LIN {X 0,Y 519.821,Z 406.729,A -85,B 0,C 180,E1 -4932.29,E2 -4932.29} C_VEL
LIN {X 0,Y 519.302,Z 420.302,A -85,B 0,C 180,E1 -4933.084,E2 -4933.084} C_VEL
LIN {X 0,Y 518.746,Z 433.349,A -85,B 0,C 180,E1 -4934.021,E2 -4934.021} C_VEL
LIN {X 0,Y 518.217,Z 445.385,A -85,B 0,C 180,E1 -4935.067,E2 -4935.067} C_VEL
LIN {X 0,Y 517.729,Z 456.81,A -85,B 0,C 180,E1 -4936.257,E2 -4936.257} C_VEL
LIN {X 0,Y 517.347,Z 466.418,A -85,B 0,C 180,E1 -4937.446,E2 -4937.446} C_VEL
LIN {X 0,Y 517.02,Z 475.827,A -85,B 0,C 180,E1 -4938.831,E2 -4938.831} C_VEL
LIN {X 0,Y 516.707,Z 483.661,A -85,B 0,C 180,E1 -4940.211,E2 -4940.211} C_VEL
LIN {X 0,Y 516.511,Z 490.966,A -85,B 0,C 180,E1 -4941.786,E2 -4941.786} C_VEL
LIN {X 0,Y 516.372,Z 497.212,A -85,B 0,C 180,E1 -4943.493,E2 -4943.493} C_VEL
LIN {X 0,Y 516.373,Z 500.263,A -85,B 0,C 180,E1 -4944.533,E2 -4944.533} C_VEL
LIN {X 0,Y 516.308,Z 503.797,A -85,B 0,C 180,E1 -4946.097,E2 -4946.097} C_VEL
LIN {X 0,Y 516.259,Z 506.138,A -85,B 0,C 180,E1 -4947.659,E2 -4947.659} C_VEL
LIN {X 0,Y 516.156,Z 507.337,A -85,B 0,C 180,E1 -4949.22,E2 -4949.22} C_VEL
LIN {X 0,Y 516.157,Z 507.356,A -85,B 0,C 180,E1 -4950.78,E2 -4950.78} C_VEL
LIN {X 0,Y 516.259,Z 506.235,A -85,B 0,C 180,E1 -4952.34,E2 -4952.34} C_VEL
LIN {X 0,Y 516.308,Z 503.97,A -85,B 0,C 180,E1 -4953.902,E2 -4953.902} C_VEL
LIN {X 0,Y 516.369,Z 500.509,A -85,B 0,C 180,E1 -4955.467,E2 -4955.467} C_VEL
LIN {X 0,Y 516.392,Z 495.769,A -85,B 0,C 180,E1 -4957.035,E2 -4957.035} C_VEL
LIN {X 0,Y 516.541,Z 489.713,A -85,B 0,C 180,E1 -4958.607,E2 -4958.607} C_VEL
LIN {X 0,Y 516.758,Z 482.087,A -85,B 0,C 180,E1 -4960.183,E2 -4960.183} C_VEL
LIN {X 0,Y 517.014,Z 473.951,A -85,B 0,C 180,E1 -4961.566,E2 -4961.566} C_VEL
LIN {X 0,Y 517.423,Z 464.143,A -85,B 0,C 180,E1 -4962.95,E2 -4962.95} C_VEL
LIN {X 0,Y 517.829,Z 454.081,A -85,B 0,C 180,E1 -4964.14,E2 -4964.14} C_VEL
LIN {X 0,Y 518.306,Z 442.542,A -85,B 0,C 180,E1 -4965.289,E2 -4965.289} C_VEL
LIN {X 0,Y 518.904,Z 430.325,A -85,B 0,C 180,E1 -4966.301,E2 -4966.301} C_VEL
LIN {X 0,Y 519.365,Z 418.57,A -85,B 0,C 180,E1 -4967.116,E2 -4967.116} C_VEL
LIN {X 0,Y 519.835,Z 404.548,A -85,B 0,C 180,E1 -4967.913,E2 -4967.913} C_VEL
LIN {X 0,Y 520.354,Z 389.292,A -85,B 0,C 180,E1 -4968.583,E2 -4968.583} C_VEL
LIN {X 0,Y 520.704,Z 373.976,A -85,B 0,C 180,E1 -4969.078,E2 -4969.078} C_VEL
LIN {X 0,Y 520.233,Z 370.683,A -85,B 0,C 180,E1 -4969.188,E2 -4969.188} C_VEL
LIN {X 0,Y 516.92,Z 358.729,A -85,B 0,C 180,E1 -4969.566,E2 -4969.566} C_VEL
LIN {X 0,Y 516.34,Z 356.363,A -85,B 0,C 180,E1 -4969.649,E2 -4969.649} C_VEL
LIN {X 0,Y 516.364,Z 353.469,A -85,B 0,C 180,E1 -4972.401,E2 -4972.401} C_VEL
LIN {X 0,Y 516.389,Z 350.798,A -85,B 0,C 180,E1 -4974.955,E2 -4974.955} C_VEL
LIN {X 0,Y 516.469,Z 348.145,A -85,B 0,C 180,E1 -4977.559,E2 -4977.559} C_VEL
LIN {X 0,Y 516.495,Z 345.564,A -85,B 0,C 180,E1 -4980.229,E2 -4980.229} C_VEL
LIN {X 0,Y 516.579,Z 342.965,A -85,B 0,C 180,E1 -4982.969,E2 -4982.969} C_VEL
LIN {X 0,Y 516.601,Z 340.308,A -85,B 0,C 180,E1 -4985.801,E2 -4985.801} C_VEL
LIN {X 0,Y 516.629,Z 337.612,A -85,B 0,C 180,E1 -4988.738,E2 -4988.738} C_VEL
LIN {X 0,Y 516.66,Z 336.757,A -85,B 0,C 180,E1 -4989.741,E2 -4989.741} C_VEL
LIN {X 0,Y 516.848,Z 336.729,A -85,B 0,C 180,E1 -4991.781,E2 -4991.781} C_VEL
LIN {X 0,Y 516.922,Z 336.72,A -85,B 0,C 180,E1 -4995.01,E2 -4995.01} C_VEL
LIN {X 0,Y 516.916,Z 336.72,A -85,B 0,C 180,E1 -4998.398,E2 -4998.398} C_VEL
LIN {X 0,Y 516.882,Z 336.724,A -85,B 0,C 180,E1 -5001.284,E2 -5001.284} C_VEL
LIN {X 0,Y 516.891,Z 336.723,A -85,B 0,C 180,E1 -5004.221,E2 -5004.221} C_VEL
LIN {X 0,Y 516.895,Z 336.72,A -85,B 0,C 180,E1 -5007.053,E2 -5007.053} C_VEL
LIN {X 0,Y 516.901,Z 336.727,A -85,B 0,C 180,E1 -5009.797,E2 -5009.797} C_VEL
LIN {X 0,Y 516.929,Z 336.716,A -85,B 0,C 180,E1 -5012.467,E2 -5012.467} C_VEL
LIN {X 0,Y 516.911,Z 336.719,A -85,B 0,C 180,E1 -5015.072,E2 -5015.072} C_VEL
LIN {X 0,Y 516.885,Z 336.721,A -85,B 0,C 180,E1 -5018.462,E2 -5018.462} C_VEL
LIN {X 0,Y 516.904,Z 336.719,A -85,B 0,C 180,E1 -5020.955,E2 -5020.955} C_VEL
LIN {X 0,Y 516.916,Z 336.724,A -85,B 0,C 180,E1 -5023.41,E2 -5023.41} C_VEL
LIN {X 0,Y 516.894,Z 336.718,A -85,B 0,C 180,E1 -5025.834,E2 -5025.834} C_VEL
LIN {X 0,Y 517.003,Z 336.71,A -85,B 0,C 180,E1 -5028.234,E2 -5028.234} C_VEL
LIN {X 0,Y 516.969,Z 336.714,A -85,B 0,C 180,E1 -5031.4,E2 -5031.4} C_VEL
LIN {X 0,Y 517.011,Z 336.709,A -85,B 0,C 180,E1 -5033.757,E2 -5033.757} C_VEL
LIN {X 0,Y 517.082,Z 336.7,A -85,B 0,C 180,E1 -5037.663,E2 -5037.663} C_VEL
LIN {X 0,Y 517.093,Z 336.698,A -85,B 0,C 180,E1 -5040.779,E2 -5040.779} C_VEL
LIN {X 0,Y 517.014,Z 336.711,A -85,B 0,C 180,E1 -5043.117,E2 -5043.117} C_VEL
LIN {X 0,Y 517.009,Z 336.713,A -85,B 0,C 180,E1 -5046.243,E2 -5046.243} C_VEL
LIN {X 0,Y 516.952,Z 336.72,A -85,B 0,C 180,E1 -5049.389,E2 -5049.389} C_VEL
LIN {X 0,Y 516.955,Z 336.715,A -85,B 0,C 180,E1 -5051.81,E2 -5051.81} C_VEL
LIN {X 0,Y 516.942,Z 336.718,A -85,B 0,C 180,E1 -5055.147,E2 -5055.147} C_VEL
LIN {X 0,Y 516.923,Z 336.72,A -85,B 0,C 180,E1 -5058.222,E2 -5058.222} C_VEL
LIN {X 0,Y 516.91,Z 336.72,A -85,B 0,C 180,E1 -5060.701,E2 -5060.701} C_VEL
LIN {X 0,Y 516.909,Z 336.722,A -85,B 0,C 180,E1 -5064.072,E2 -5064.072} C_VEL
LIN {X 0,Y 516.924,Z 336.72,A -85,B 0,C 180,E1 -5066.658,E2 -5066.658} C_VEL
LIN {X 0,Y 516.918,Z 336.722,A -85,B 0,C 180,E1 -5069.526,E2 -5069.526} C_VEL
LIN {X 0,Y 516.899,Z 336.724,A -85,B 0,C 180,E1 -5072.544,E2 -5072.544} C_VEL
LIN {X 0,Y 516.881,Z 336.728,A -85,B 0,C 180,E1 -5075.333,E2 -5075.333} C_VEL
LIN {X 0,Y 516.88,Z 336.727,A -85,B 0,C 180,E1 -5077.944,E2 -5077.944} C_VEL
LIN {X 0,Y 516.884,Z 336.726,A -85,B 0,C 180,E1 -5080.742,E2 -5080.742} C_VEL
LIN {X 0,Y 516.882,Z 336.724,A -85,B 0,C 180,E1 -5082.831,E2 -5082.831} C_VEL
LIN {X 0,Y 516.924,Z 336.727,A -85,B 0,C 180,E1 -5085.011,E2 -5085.011} C_VEL
LIN {X 0,Y 517.783,Z 342.257,A -85,B 0,C 180,E1 -5087.789,E2 -5087.789} C_VEL
LIN {X 0,Y 517.985,Z 345.864,A -85,B 0,C 180,E1 -5089.447,E2 -5089.447} C_VEL
LIN {X 0,Y 517.741,Z 352.598,A -85,B 0,C 180,E1 -5092.35,E2 -5092.35} C_VEL
LIN {X 0,Y 517.609,Z 357.962,A -85,B 0,C 180,E1 -5094.554,E2 -5094.554} C_VEL
LIN {X 0,Y 517.413,Z 365.096,A -85,B 0,C 180,E1 -5097.367,E2 -5097.367} C_VEL
LIN {X 0,Y 517.242,Z 373.131,A -85,B 0,C 180,E1 -5100.412,E2 -5100.412} C_VEL
LIN {X 0,Y 517.066,Z 381.047,A -85,B 0,C 180,E1 -5103.35,E2 -5103.35} C_VEL
LIN {X 0,Y 516.871,Z 389.351,A -85,B 0,C 180,E1 -5106.352,E2 -5106.352} C_VEL
LIN {X 0,Y 516.77,Z 397.674,A -85,B 0,C 180,E1 -5109.293,E2 -5109.293} C_VEL
LIN {X 0,Y 516.703,Z 400.834,A -85,B 0,C 180,E1 -5110.381,E2 -5110.381} C_VEL
LIN {X 0,Y 520.44,Z 417.085,A -85,B 0,C 180,E1 -5110.825,E2 -5110.825} C_VEL
LIN {X 0,Y 520.664,Z 420.573,A -85,B 0,C 180,E1 -5110.919,E2 -5110.919} C_VEL
LIN {X 0,Y 520.288,Z 434.02,A -85,B 0,C 180,E1 -5111.32,E2 -5111.32} C_VEL
LIN {X 0,Y 519.885,Z 449.136,A -85,B 0,C 180,E1 -5111.936,E2 -5111.936} C_VEL
LIN {X 0,Y 519.372,Z 463.303,A -85,B 0,C 180,E1 -5112.681,E2 -5112.681} C_VEL
LIN {X 0,Y 518.84,Z 477.112,A -85,B 0,C 180,E1 -5113.585,E2 -5113.585} C_VEL
LIN {X 0,Y 518.397,Z 489.137,A -85,B 0,C 180,E1 -5114.542,E2 -5114.542} C_VEL
LIN {X 0,Y 517.857,Z 500.982,A -85,B 0,C 180,E1 -5115.66,E2 -5115.66} C_VEL
LIN {X 0,Y 517.47,Z 511.579,A -85,B 0,C 180,E1 -5116.851,E2 -5116.851} C_VEL
LIN {X 0,Y 517.012,Z 521.94,A -85,B 0,C 180,E1 -5118.235,E2 -5118.235} C_VEL
LIN {X 0,Y 516.89,Z 529.417,A -85,B 0,C 180,E1 -5119.423,E2 -5119.423} C_VEL
LIN {X 0,Y 516.637,Z 535.751,A -85,B 0,C 180,E1 -5120.605,E2 -5120.605} C_VEL
LIN {X 0,Y 516.462,Z 542.701,A -85,B 0,C 180,E1 -5122.179,E2 -5122.179} C_VEL
LIN {X 0,Y 516.36,Z 548.163,A -85,B 0,C 180,E1 -5123.749,E2 -5123.749} C_VEL
LIN {X 0,Y 516.238,Z 552.291,A -85,B 0,C 180,E1 -5125.315,E2 -5125.315} C_VEL
LIN {X 0,Y 516.272,Z 555.184,A -85,B 0,C 180,E1 -5126.879,E2 -5126.879} C_VEL
LIN {X 0,Y 516.189,Z 556.909,A -85,B 0,C 180,E1 -5128.44,E2 -5128.44} C_VEL
LIN {X 0,Y 516.151,Z 557.5,A -85,B 0,C 180,E1 -5130,E2 -5130} C_VEL
LIN {X 0,Y 516.189,Z 556.906,A -85,B 0,C 180,E1 -5131.561,E2 -5131.561} C_VEL
LIN {X 0,Y 516.272,Z 555.178,A -85,B 0,C 180,E1 -5133.122,E2 -5133.122} C_VEL
LIN {X 0,Y 516.238,Z 552.287,A -85,B 0,C 180,E1 -5134.686,E2 -5134.686} C_VEL
LIN {X 0,Y 516.376,Z 548.164,A -85,B 0,C 180,E1 -5136.251,E2 -5136.251} C_VEL
LIN {X 0,Y 516.463,Z 542.699,A -85,B 0,C 180,E1 -5137.821,E2 -5137.821} C_VEL
LIN {X 0,Y 516.638,Z 535.741,A -85,B 0,C 180,E1 -5139.395,E2 -5139.395} C_VEL
LIN {X 0,Y 516.911,Z 528.287,A -85,B 0,C 180,E1 -5140.775,E2 -5140.775} C_VEL
LIN {X 0,Y 517.138,Z 519.473,A -85,B 0,C 180,E1 -5142.121,E2 -5142.121} C_VEL
LIN {X 0,Y 517.536,Z 509.929,A -85,B 0,C 180,E1 -5143.348,E2 -5143.348} C_VEL
LIN {X 0,Y 517.917,Z 499.008,A -85,B 0,C 180,E1 -5144.539,E2 -5144.539} C_VEL
LIN {X 0,Y 518.445,Z 487.256,A -85,B 0,C 180,E1 -5145.617,E2 -5145.617} C_VEL
LIN {X 0,Y 518.952,Z 474.093,A -85,B 0,C 180,E1 -5146.624,E2 -5146.624} C_VEL
LIN {X 0,Y 519.491,Z 459.731,A -85,B 0,C 180,E1 -5147.519,E2 -5147.519} C_VEL
LIN {X 0,Y 520.048,Z 444.783,A -85,B 0,C 180,E1 -5148.254,E2 -5148.254} C_VEL
LIN {X 0,Y 520.425,Z 429.866,A -85,B 0,C 180,E1 -5148.814,E2 -5148.814} C_VEL
LIN {X 0,Y 520.592,Z 417.655,A -85,B 0,C 180,E1 -5149.157,E2 -5149.157} C_VEL
LIN {X 0,Y 516.706,Z 400.814,A -85,B 0,C 180,E1 -5149.626,E2 -5149.626} C_VEL
LIN {X 0,Y 516.833,Z 392.896,A -85,B 0,C 180,E1 -5152.38,E2 -5152.38} C_VEL
LIN {X 0,Y 517.025,Z 383.43,A -85,B 0,C 180,E1 -5155.784,E2 -5155.784} C_VEL
LIN {X 0,Y 517.201,Z 375.092,A -85,B 0,C 180,E1 -5158.842,E2 -5158.842} C_VEL
LIN {X 0,Y 517.373,Z 366.731,A -85,B 0,C 180,E1 -5161.991,E2 -5161.991} C_VEL
LIN {X 0,Y 517.517,Z 359.618,A -85,B 0,C 180,E1 -5164.776,E2 -5164.776} C_VEL
LIN {X 0,Y 517.741,Z 352.555,A -85,B 0,C 180,E1 -5167.651,E2 -5167.651} C_VEL
LIN {X 0,Y 517.907,Z 346.893,A -85,B 0,C 180,E1 -5170.085,E2 -5170.085} C_VEL
LIN {X 0,Y 517.896,Z 343.265,A -85,B 0,C 180,E1 -5171.724,E2 -5171.724} C_VEL
LIN {X 0,Y 517.082,Z 337.701,A -85,B 0,C 180,E1 -5174.475,E2 -5174.475} C_VEL
LIN {X 0,Y 516.916,Z 336.724,A -85,B 0,C 180,E1 -5175.009,E2 -5175.009} C_VEL
LIN {X 0,Y 516.915,Z 336.723,A -85,B 0,C 180,E1 -5178.399,E2 -5178.399} C_VEL
LIN {X 0,Y 516.884,Z 336.727,A -85,B 0,C 180,E1 -5181.284,E2 -5181.284} C_VEL
LIN {X 0,Y 516.894,Z 336.725,A -85,B 0,C 180,E1 -5184.222,E2 -5184.222} C_VEL
LIN {X 0,Y 516.897,Z 336.723,A -85,B 0,C 180,E1 -5187.053,E2 -5187.053} C_VEL
LIN {X 0,Y 516.895,Z 336.724,A -85,B 0,C 180,E1 -5189.797,E2 -5189.797} C_VEL
LIN {X 0,Y 516.931,Z 336.723,A -85,B 0,C 180,E1 -5192.468,E2 -5192.468} C_VEL
LIN {X 0,Y 516.911,Z 336.722,A -85,B 0,C 180,E1 -5195.072,E2 -5195.072} C_VEL
LIN {X 0,Y 516.889,Z 336.728,A -85,B 0,C 180,E1 -5198.463,E2 -5198.463} C_VEL
LIN {X 0,Y 516.906,Z 336.721,A -85,B 0,C 180,E1 -5200.955,E2 -5200.955} C_VEL
LIN {X 0,Y 516.917,Z 336.722,A -85,B 0,C 180,E1 -5203.41,E2 -5203.41} C_VEL
LIN {X 0,Y 516.899,Z 336.725,A -85,B 0,C 180,E1 -5205.834,E2 -5205.834} C_VEL
LIN {X 0,Y 516.969,Z 336.714,A -85,B 0,C 180,E1 -5208.234,E2 -5208.234} C_VEL
LIN {X 0,Y 516.972,Z 336.713,A -85,B 0,C 180,E1 -5211.4,E2 -5211.4} C_VEL
LIN {X 0,Y 517.013,Z 336.712,A -85,B 0,C 180,E1 -5213.757,E2 -5213.757} C_VEL
LIN {X 0,Y 517.087,Z 336.698,A -85,B 0,C 180,E1 -5217.663,E2 -5217.663} C_VEL
LIN {X 0,Y 517.098,Z 336.697,A -85,B 0,C 180,E1 -5220.779,E2 -5220.779} C_VEL
LIN {X 0,Y 517.017,Z 336.708,A -85,B 0,C 180,E1 -5223.117,E2 -5223.117} C_VEL
LIN {X 0,Y 517.015,Z 336.707,A -85,B 0,C 180,E1 -5226.243,E2 -5226.243} C_VEL
LIN {X 0,Y 516.957,Z 336.715,A -85,B 0,C 180,E1 -5229.389,E2 -5229.389} C_VEL
LIN {X 0,Y 516.956,Z 336.714,A -85,B 0,C 180,E1 -5231.807,E2 -5231.807} C_VEL
LIN {X 0,Y 516.948,Z 336.719,A -85,B 0,C 180,E1 -5235.146,E2 -5235.146} C_VEL
LIN {X 0,Y 516.929,Z 336.719,A -85,B 0,C 180,E1 -5238.222,E2 -5238.222} C_VEL
LIN {X 0,Y 516.916,Z 336.711,A -85,B 0,C 180,E1 -5240.701,E2 -5240.701} C_VEL
LIN {X 0,Y 516.894,Z 336.726,A -85,B 0,C 180,E1 -5244.073,E2 -5244.073} C_VEL
LIN {X 0,Y 516.928,Z 336.714,A -85,B 0,C 180,E1 -5246.658,E2 -5246.658} C_VEL
LIN {X 0,Y 516.915,Z 336.719,A -85,B 0,C 180,E1 -5249.524,E2 -5249.524} C_VEL
LIN {X 0,Y 516.899,Z 336.719,A -85,B 0,C 180,E1 -5252.543,E2 -5252.543} C_VEL
LIN {X 0,Y 516.883,Z 336.724,A -85,B 0,C 180,E1 -5255.332,E2 -5255.332} C_VEL
LIN {X 0,Y 516.885,Z 336.729,A -85,B 0,C 180,E1 -5257.943,E2 -5257.943} C_VEL
LIN {X 0,Y 516.888,Z 336.727,A -85,B 0,C 180,E1 -5260.741,E2 -5260.741} C_VEL
LIN {X 0,Y 516.887,Z 336.726,A -85,B 0,C 180,E1 -5262.831,E2 -5262.831} C_VEL
LIN {X 0,Y 516.926,Z 336.72,A -85,B 0,C 180,E1 -5265.01,E2 -5265.01} C_VEL
LIN {X 0,Y 516.851,Z 336.731,A -85,B 0,C 180,E1 -5268.218,E2 -5268.218} C_VEL
LIN {X 0,Y 516.672,Z 336.776,A -85,B 0,C 180,E1 -5270.292,E2 -5270.292} C_VEL
LIN {X 0,Y 515.975,Z 337.328,A -85,B 0,C 180,E1 -5270.939,E2 -5270.939} C_VEL
LIN {X 0,Y 513.098,Z 338.557,A -85,B 0,C 180,E1 -5271.987,E2 -5271.987} C_VEL
LIN {X 0,Y 510.678,Z 339.577,A -85,B 0,C 180,E1 -5272.83,E2 -5272.83} C_VEL
LIN {X 0,Y 509.635,Z 340.277,A -85,B 0,C 180,E1 -5273.482,E2 -5273.482} C_VEL
LIN {X 0,Y 509.547,Z 340.487,A -85,B 0,C 180,E1 -5273.703,E2 -5273.703} C_VEL
LIN {X 0,Y 509.517,Z 343.074,A -85,B 0,C 180,E1 -5276.513,E2 -5276.513} C_VEL
LIN {X 0,Y 509.437,Z 345.693,A -85,B 0,C 180,E1 -5279.307,E2 -5279.307} C_VEL
LIN {X 0,Y 509.404,Z 348.283,A -85,B 0,C 180,E1 -5282.025,E2 -5282.025} C_VEL
LIN {X 0,Y 509.356,Z 350.915,A -85,B 0,C 180,E1 -5284.676,E2 -5284.676} C_VEL
LIN {X 0,Y 509.299,Z 353.973,A -85,B 0,C 180,E1 -5287.602,E2 -5287.602} C_VEL
LIN {X 0,Y 509.284,Z 356.802,A -85,B 0,C 180,E1 -5290.177,E2 -5290.177} C_VEL
LIN {X 0,Y 513.395,Z 371.414,A -85,B 0,C 180,E1 -5290.646,E2 -5290.646} C_VEL
LIN {X 0,Y 513.96,Z 374.193,A -85,B 0,C 180,E1 -5290.748,E2 -5290.748} C_VEL
LIN {X 0,Y 513.663,Z 388.561,A -85,B 0,C 180,E1 -5291.213,E2 -5291.213} C_VEL
LIN {X 0,Y 513.16,Z 403.143,A -85,B 0,C 180,E1 -5291.846,E2 -5291.846} C_VEL
LIN {X 0,Y 512.634,Z 417.516,A -85,B 0,C 180,E1 -5292.651,E2 -5292.651} C_VEL
LIN {X 0,Y 512.067,Z 430.567,A -85,B 0,C 180,E1 -5293.556,E2 -5293.556} C_VEL
LIN {X 0,Y 511.549,Z 441.99,A -85,B 0,C 180,E1 -5294.507,E2 -5294.507} C_VEL
LIN {X 0,Y 510.97,Z 453.632,A -85,B 0,C 180,E1 -5295.666,E2 -5295.666} C_VEL
LIN {X 0,Y 510.518,Z 463.777,A -85,B 0,C 180,E1 -5296.871,E2 -5296.871} C_VEL
LIN {X 0,Y 510.087,Z 473.286,A -85,B 0,C 180,E1 -5298.211,E2 -5298.211} C_VEL
LIN {X 0,Y 509.828,Z 480.826,A -85,B 0,C 180,E1 -5299.475,E2 -5299.475} C_VEL
LIN {X 0,Y 509.584,Z 487.865,A -85,B 0,C 180,E1 -5300.874,E2 -5300.874} C_VEL
LIN {X 0,Y 509.39,Z 494.393,A -85,B 0,C 180,E1 -5302.468,E2 -5302.468} C_VEL
LIN {X 0,Y 509.313,Z 499.494,A -85,B 0,C 180,E1 -5304.059,E2 -5304.059} C_VEL
LIN {X 0,Y 509.159,Z 502.438,A -85,B 0,C 180,E1 -5305.249,E2 -5305.249} C_VEL
LIN {X 0,Y 509.188,Z 505.316,A -85,B 0,C 180,E1 -5306.835,E2 -5306.835} C_VEL
LIN {X 0,Y 509.11,Z 507.057,A -85,B 0,C 180,E1 -5308.418,E2 -5308.418} C_VEL
LIN {X 0,Y 509.063,Z 507.667,A -85,B 0,C 180,E1 -5310,E2 -5310} C_VEL
LIN {X 0,Y 509.111,Z 507.113,A -85,B 0,C 180,E1 -5311.582,E2 -5311.582} C_VEL
LIN {X 0,Y 509.189,Z 505.448,A -85,B 0,C 180,E1 -5313.165,E2 -5313.165} C_VEL
LIN {X 0,Y 509.158,Z 502.641,A -85,B 0,C 180,E1 -5314.75,E2 -5314.75} C_VEL
LIN {X 0,Y 509.26,Z 498.613,A -85,B 0,C 180,E1 -5316.338,E2 -5316.338} C_VEL
LIN {X 0,Y 509.412,Z 493.269,A -85,B 0,C 180,E1 -5317.93,E2 -5317.93} C_VEL
LIN {X 0,Y 509.614,Z 486.458,A -85,B 0,C 180,E1 -5319.525,E2 -5319.525} C_VEL
LIN {X 0,Y 509.96,Z 477.948,A -85,B 0,C 180,E1 -5321.124,E2 -5321.124} C_VEL
LIN {X 0,Y 510.285,Z 468.902,A -85,B 0,C 180,E1 -5322.528,E2 -5322.528} C_VEL
LIN {X 0,Y 510.698,Z 459.668,A -85,B 0,C 180,E1 -5323.732,E2 -5323.732} C_VEL
LIN {X 0,Y 511.237,Z 447.728,A -85,B 0,C 180,E1 -5325.039,E2 -5325.039} C_VEL
LIN {X 0,Y 511.86,Z 435.522,A -85,B 0,C 180,E1 -5326.142,E2 -5326.142} C_VEL
LIN {X 0,Y 512.447,Z 422.046,A -85,B 0,C 180,E1 -5327.149,E2 -5327.149} C_VEL
LIN {X 0,Y 512.959,Z 408.785,A -85,B 0,C 180,E1 -5327.955,E2 -5327.955} C_VEL
LIN {X 0,Y 513.493,Z 394.989,A -85,B 0,C 180,E1 -5328.619,E2 -5328.619} C_VEL
LIN {X 0,Y 513.869,Z 380.906,A -85,B 0,C 180,E1 -5329.142,E2 -5329.142} C_VEL
LIN {X 0,Y 513.814,Z 373.203,A -85,B 0,C 180,E1 -5329.376,E2 -5329.376} C_VEL
LIN {X 0,Y 510.626,Z 361.408,A -85,B 0,C 180,E1 -5329.776,E2 -5329.776} C_VEL
LIN {X 0,Y 509.297,Z 356.686,A -85,B 0,C 180,E1 -5329.92,E2 -5329.92} C_VEL
LIN {X 0,Y 509.289,Z 353.731,A -85,B 0,C 180,E1 -5332.73,E2 -5332.73} C_VEL
LIN {X 0,Y 509.353,Z 351.009,A -85,B 0,C 180,E1 -5335.323,E2 -5335.323} C_VEL
LIN {X 0,Y 509.388,Z 348.368,A -85,B 0,C 180,E1 -5337.993,E2 -5337.993} C_VEL
LIN {X 0,Y 509.476,Z 345.302,A -85,B 0,C 180,E1 -5341.211,E2 -5341.211} C_VEL
LIN {X 0,Y 509.541,Z 342.55,A -85,B 0,C 180,E1 -5344.15,E2 -5344.15} C_VEL
LIN {X 0,Y 509.562,Z 340.045,A -85,B 0,C 180,E1 -5346.875,E2 -5346.875} C_VEL
LIN {X 0,Y 509.589,Z 337.733,A -85,B 0,C 180,E1 -5349.437,E2 -5349.437} C_VEL
LIN {X 0,Y 509.803,Z 337.605,A -85,B 0,C 180,E1 -5351.89,E2 -5351.89} C_VEL
LIN {X 0,Y 509.856,Z 337.603,A -85,B 0,C 180,E1 -5354.668,E2 -5354.668} C_VEL
LIN {X 0,Y 509.857,Z 337.6,A -85,B 0,C 180,E1 -5358.103,E2 -5358.103} C_VEL
LIN {X 0,Y 509.847,Z 337.605,A -85,B 0,C 180,E1 -5360.647,E2 -5360.647} C_VEL
LIN {X 0,Y 509.836,Z 337.606,A -85,B 0,C 180,E1 -5363.648,E2 -5363.648} C_VEL
LIN {X 0,Y 509.861,Z 337.599,A -85,B 0,C 180,E1 -5366.539,E2 -5366.539} C_VEL
LIN {X 0,Y 509.85,Z 337.6,A -85,B 0,C 180,E1 -5369.334,E2 -5369.334} C_VEL
LIN {X 0,Y 509.894,Z 337.59,A -85,B 0,C 180,E1 -5372.054,E2 -5372.054} C_VEL
LIN {X 0,Y 509.877,Z 337.597,A -85,B 0,C 180,E1 -5374.704,E2 -5374.704} C_VEL
LIN {X 0,Y 509.855,Z 337.601,A -85,B 0,C 180,E1 -5377.449,E2 -5377.449} C_VEL
LIN {X 0,Y 509.915,Z 337.583,A -85,B 0,C 180,E1 -5379.845,E2 -5379.845} C_VEL
LIN {X 0,Y 509.886,Z 337.597,A -85,B 0,C 180,E1 -5383.175,E2 -5383.175} C_VEL
LIN {X 0,Y 509.863,Z 337.593,A -85,B 0,C 180,E1 -5385.634,E2 -5385.634} C_VEL
LIN {X 0,Y 509.921,Z 337.589,A -85,B 0,C 180,E1 -5388.875,E2 -5388.875} C_VEL
LIN {X 0,Y 509.95,Z 337.587,A -85,B 0,C 180,E1 -5392.078,E2 -5392.078} C_VEL
LIN {X 0,Y 509.982,Z 337.585,A -85,B 0,C 180,E1 -5394.464,E2 -5394.464} C_VEL
LIN {X 0,Y 510.053,Z 337.576,A -85,B 0,C 180,E1 -5397.631,E2 -5397.631} C_VEL
LIN {X 0,Y 510.063,Z 337.574,A -85,B 0,C 180,E1 -5400.789,E2 -5400.789} C_VEL
LIN {X 0,Y 509.956,Z 337.59,A -85,B 0,C 180,E1 -5403.16,E2 -5403.16} C_VEL
LIN {X 0,Y 509.977,Z 337.589,A -85,B 0,C 180,E1 -5406.33,E2 -5406.33} C_VEL
LIN {X 0,Y 509.914,Z 337.592,A -85,B 0,C 180,E1 -5408.72,E2 -5408.72} C_VEL
LIN {X 0,Y 509.903,Z 337.594,A -85,B 0,C 180,E1 -5411.932,E2 -5411.932} C_VEL
LIN {X 0,Y 509.891,Z 337.597,A -85,B 0,C 180,E1 -5415.242,E2 -5415.242} C_VEL
LIN {X 0,Y 509.886,Z 337.595,A -85,B 0,C 180,E1 -5418.001,E2 -5418.001} C_VEL
LIN {X 0,Y 509.848,Z 337.6,A -85,B 0,C 180,E1 -5421.002,E2 -5421.002} C_VEL
LIN {X 0,Y 509.835,Z 337.603,A -85,B 0,C 180,E1 -5423.563,E2 -5423.563} C_VEL
LIN {X 0,Y 509.91,Z 337.596,A -85,B 0,C 180,E1 -5426.379,E2 -5426.379} C_VEL
LIN {X 0,Y 509.879,Z 337.599,A -85,B 0,C 180,E1 -5428.844,E2 -5428.844} C_VEL
LIN {X 0,Y 509.824,Z 337.604,A -85,B 0,C 180,E1 -5431.59,E2 -5431.59} C_VEL
LIN {X 0,Y 509.852,Z 337.601,A -85,B 0,C 180,E1 -5434.413,E2 -5434.413} C_VEL
LIN {X 0,Y 509.818,Z 337.605,A -85,B 0,C 180,E1 -5437.341,E2 -5437.341} C_VEL
LIN {X 0,Y 509.837,Z 337.604,A -85,B 0,C 180,E1 -5440.382,E2 -5440.382} C_VEL
LIN {X 0,Y 509.822,Z 337.604,A -85,B 0,C 180,E1 -5443.063,E2 -5443.063} C_VEL
LIN {X 0,Y 509.873,Z 337.71,A -85,B 0,C 180,E1 -5444.756,E2 -5444.756} C_VEL
LIN {X 0,Y 510.778,Z 343.299,A -85,B 0,C 180,E1 -5447.608,E2 -5447.608} C_VEL
LIN {X 0,Y 511.015,Z 346.574,A -85,B 0,C 180,E1 -5449.149,E2 -5449.149} C_VEL
LIN {X 0,Y 510.812,Z 352.471,A -85,B 0,C 180,E1 -5451.748,E2 -5451.748} C_VEL
LIN {X 0,Y 510.597,Z 359.462,A -85,B 0,C 180,E1 -5454.683,E2 -5454.683} C_VEL
LIN {X 0,Y 510.364,Z 367.762,A -85,B 0,C 180,E1 -5457.984,E2 -5457.984} C_VEL
LIN {X 0,Y 510.181,Z 376.111,A -85,B 0,C 180,E1 -5461.175,E2 -5461.175} C_VEL
LIN {X 0,Y 509.947,Z 384.411,A -85,B 0,C 180,E1 -5464.271,E2 -5464.271} C_VEL
LIN {X 0,Y 509.772,Z 393.14,A -85,B 0,C 180,E1 -5467.473,E2 -5467.473} C_VEL
LIN {X 0,Y 509.643,Z 400.435,A -85,B 0,C 180,E1 -5470.087,E2 -5470.087} C_VEL
LIN {X 0,Y 513.688,Z 418.149,A -85,B 0,C 180,E1 -5470.595,E2 -5470.595} C_VEL
LIN {X 0,Y 513.921,Z 420.916,A -85,B 0,C 180,E1 -5470.679,E2 -5470.679} C_VEL
LIN {X 0,Y 513.527,Z 434.316,A -85,B 0,C 180,E1 -5471.088,E2 -5471.088} C_VEL
LIN {X 0,Y 513.108,Z 448.787,A -85,B 0,C 180,E1 -5471.689,E2 -5471.689} C_VEL
LIN {X 0,Y 512.558,Z 462.953,A -85,B 0,C 180,E1 -5472.443,E2 -5472.443} C_VEL
LIN {X 0,Y 511.967,Z 476.618,A -85,B 0,C 180,E1 -5473.348,E2 -5473.348} C_VEL
LIN {X 0,Y 511.437,Z 489.463,A -85,B 0,C 180,E1 -5474.385,E2 -5474.385} C_VEL
LIN {X 0,Y 510.905,Z 500.63,A -85,B 0,C 180,E1 -5475.461,E2 -5475.461} C_VEL
LIN {X 0,Y 510.476,Z 511.227,A -85,B 0,C 180,E1 -5476.668,E2 -5476.668} C_VEL
LIN {X 0,Y 510.001,Z 521.589,A -85,B 0,C 180,E1 -5478.071,E2 -5478.071} C_VEL
LIN {X 0,Y 509.786,Z 530.216,A -85,B 0,C 180,E1 -5479.475,E2 -5479.475} C_VEL
LIN {X 0,Y 509.516,Z 537.391,A -85,B 0,C 180,E1 -5480.873,E2 -5480.873} C_VEL
LIN {X 0,Y 509.351,Z 544.053,A -85,B 0,C 180,E1 -5482.468,E2 -5482.468} C_VEL
LIN {X 0,Y 509.275,Z 549.268,A -85,B 0,C 180,E1 -5484.06,E2 -5484.06} C_VEL
LIN {X 0,Y 509.158,Z 552.277,A -85,B 0,C 180,E1 -5485.25,E2 -5485.25} C_VEL
LIN {X 0,Y 509.188,Z 555.183,A -85,B 0,C 180,E1 -5486.835,E2 -5486.835} C_VEL
LIN {X 0,Y 509.11,Z 556.909,A -85,B 0,C 180,E1 -5488.418,E2 -5488.418} C_VEL
LIN {X 0,Y 509.062,Z 557.5,A -85,B 0,C 180,E1 -5490,E2 -5490} C_VEL
LIN {X 0,Y 509.11,Z 556.906,A -85,B 0,C 180,E1 -5491.582,E2 -5491.582} C_VEL
LIN {X 0,Y 509.188,Z 555.177,A -85,B 0,C 180,E1 -5493.165,E2 -5493.165} C_VEL
LIN {X 0,Y 509.159,Z 552.274,A -85,B 0,C 180,E1 -5494.751,E2 -5494.751} C_VEL
LIN {X 0,Y 509.306,Z 548.094,A -85,B 0,C 180,E1 -5496.338,E2 -5496.338} C_VEL
LIN {X 0,Y 509.385,Z 542.545,A -85,B 0,C 180,E1 -5497.931,E2 -5497.931} C_VEL
LIN {X 0,Y 509.546,Z 535.488,A -85,B 0,C 180,E1 -5499.527,E2 -5499.527} C_VEL
LIN {X 0,Y 509.905,Z 526.716,A -85,B 0,C 180,E1 -5501.126,E2 -5501.126} C_VEL
LIN {X 0,Y 510.201,Z 517.396,A -85,B 0,C 180,E1 -5502.531,E2 -5502.531} C_VEL
LIN {X 0,Y 510.607,Z 507.929,A -85,B 0,C 180,E1 -5503.735,E2 -5503.735} C_VEL
LIN {X 0,Y 511.103,Z 495.661,A -85,B 0,C 180,E1 -5505.043,E2 -5505.043} C_VEL
LIN {X 0,Y 511.718,Z 483.163,A -85,B 0,C 180,E1 -5506.148,E2 -5506.148} C_VEL
LIN {X 0,Y 512.212,Z 470.869,A -85,B 0,C 180,E1 -5507.055,E2 -5507.055} C_VEL
LIN {X 0,Y 512.749,Z 457.605,A -85,B 0,C 180,E1 -5507.86,E2 -5507.86} C_VEL
LIN {X 0,Y 513.305,Z 443.025,A -85,B 0,C 180,E1 -5508.566,E2 -5508.566} C_VEL
LIN {X 0,Y 513.713,Z 428.753,A -85,B 0,C 180,E1 -5509.095,E2 -5509.095} C_VEL
LIN {X 0,Y 513.847,Z 418.782,A -85,B 0,C 180,E1 -5509.384,E2 -5509.384} C_VEL
LIN {X 0,Y 509.995,Z 402.5,A -85,B 0,C 180,E1 -5509.859,E2 -5509.859} C_VEL
LIN {X 0,Y 509.622,Z 400.449,A -85,B 0,C 180,E1 -5509.909,E2 -5509.909} C_VEL
LIN {X 0,Y 509.749,Z 392.638,A -85,B 0,C 180,E1 -5512.709,E2 -5512.709} C_VEL
LIN {X 0,Y 509.96,Z 384.4,A -85,B 0,C 180,E1 -5515.729,E2 -5515.729} C_VEL
LIN {X 0,Y 510.179,Z 376.071,A -85,B 0,C 180,E1 -5518.826,E2 -5518.826} C_VEL
LIN {X 0,Y 510.365,Z 367.721,A -85,B 0,C 180,E1 -5522.017,E2 -5522.017} C_VEL
LIN {X 0,Y 510.591,Z 359.445,A -85,B 0,C 180,E1 -5525.318,E2 -5525.318} C_VEL
LIN {X 0,Y 510.811,Z 352.184,A -85,B 0,C 180,E1 -5528.35,E2 -5528.35} C_VEL
LIN {X 0,Y 510.968,Z 346.552,A -85,B 0,C 180,E1 -5530.845,E2 -5530.845} C_VEL
LIN {X 0,Y 510.777,Z 343.268,A -85,B 0,C 180,E1 -5532.393,E2 -5532.393} C_VEL
LIN {X 0,Y 509.853,Z 337.599,A -85,B 0,C 180,E1 -5535.332,E2 -5535.332} C_VEL
LIN {X 0,Y 509.857,Z 337.603,A -85,B 0,C 180,E1 -5538.575,E2 -5538.575} C_VEL
LIN {X 0,Y 509.854,Z 337.605,A -85,B 0,C 180,E1 -5541.787,E2 -5541.787} C_VEL
LIN {X 0,Y 509.849,Z 337.605,A -85,B 0,C 180,E1 -5544.624,E2 -5544.624} C_VEL
LIN {X 0,Y 509.863,Z 337.601,A -85,B 0,C 180,E1 -5547.481,E2 -5547.481} C_VEL
LIN {X 0,Y 509.861,Z 337.599,A -85,B 0,C 180,E1 -5550.274,E2 -5550.274} C_VEL
LIN {X 0,Y 509.888,Z 337.596,A -85,B 0,C 180,E1 -5552.945,E2 -5552.945} C_VEL
LIN {X 0,Y 509.867,Z 337.602,A -85,B 0,C 180,E1 -5555.574,E2 -5555.574} C_VEL
LIN {X 0,Y 509.854,Z 337.6,A -85,B 0,C 180,E1 -5558.999,E2 -5558.999} C_VEL
LIN {X 0,Y 509.892,Z 337.596,A -85,B 0,C 180,E1 -5561.999,E2 -5561.999} C_VEL
LIN {X 0,Y 509.914,Z 337.596,A -85,B 0,C 180,E1 -5564.819,E2 -5564.819} C_VEL
LIN {X 0,Y 509.905,Z 337.595,A -85,B 0,C 180,E1 -5568.124,E2 -5568.124} C_VEL
LIN {X 0,Y 509.918,Z 337.592,A -85,B 0,C 180,E1 -5571.28,E2 -5571.28} C_VEL
LIN {X 0,Y 509.981,Z 337.588,A -85,B 0,C 180,E1 -5573.671,E2 -5573.671} C_VEL
LIN {X 0,Y 510.058,Z 337.574,A -85,B 0,C 180,E1 -5577.631,E2 -5577.631} C_VEL
LIN {X 0,Y 510.068,Z 337.572,A -85,B 0,C 180,E1 -5580.79,E2 -5580.79} C_VEL
LIN {X 0,Y 509.959,Z 337.587,A -85,B 0,C 180,E1 -5583.16,E2 -5583.16} C_VEL
LIN {X 0,Y 509.984,Z 337.583,A -85,B 0,C 180,E1 -5586.33,E2 -5586.33} C_VEL
LIN {X 0,Y 509.92,Z 337.594,A -85,B 0,C 180,E1 -5588.72,E2 -5588.72} C_VEL
LIN {X 0,Y 509.908,Z 337.589,A -85,B 0,C 180,E1 -5591.932,E2 -5591.932} C_VEL
LIN {X 0,Y 509.898,Z 337.596,A -85,B 0,C 180,E1 -5595.242,E2 -5595.242} C_VEL
LIN {X 0,Y 509.892,Z 337.598,A -85,B 0,C 180,E1 -5598.001,E2 -5598.001} C_VEL
LIN {X 0,Y 509.854,Z 337.593,A -85,B 0,C 180,E1 -5601.002,E2 -5601.002} C_VEL
LIN {X 0,Y 509.826,Z 337.602,A -85,B 0,C 180,E1 -5603.564,E2 -5603.564} C_VEL
LIN {X 0,Y 509.915,Z 337.587,A -85,B 0,C 180,E1 -5606.378,E2 -5606.378} C_VEL
LIN {X 0,Y 509.88,Z 337.598,A -85,B 0,C 180,E1 -5608.844,E2 -5608.844} C_VEL
LIN {X 0,Y 509.824,Z 337.606,A -85,B 0,C 180,E1 -5611.59,E2 -5611.59} C_VEL
LIN {X 0,Y 509.855,Z 337.596,A -85,B 0,C 180,E1 -5614.413,E2 -5614.413} C_VEL
LIN {X 0,Y 509.823,Z 337.604,A -85,B 0,C 180,E1 -5617.34,E2 -5617.34} C_VEL
LIN {X 0,Y 509.841,Z 337.602,A -85,B 0,C 180,E1 -5620.382,E2 -5620.382} C_VEL
LIN {X 0,Y 509.827,Z 337.604,A -85,B 0,C 180,E1 -5623.062,E2 -5623.062} C_VEL
LIN {X 0,Y 509.834,Z 337.606,A -85,B 0,C 180,E1 -5625.792,E2 -5625.792} C_VEL
LIN {X 0,Y 509.777,Z 337.615,A -85,B 0,C 180,E1 -5628.566,E2 -5628.566} C_VEL
LIN {X 0,Y 509.601,Z 337.7,A -85,B 0,C 180,E1 -5630.625,E2 -5630.625} C_VEL
LIN {X 0,Y 509.547,Z 340.487,A -85,B 0,C 180,E1 -5633.703,E2 -5633.703} C_VEL
LIN {X 0,Y 508.875,Z 341.159,A -85,B 0,C 180,E1 -5634.359,E2 -5634.359} C_VEL
LIN {X 0,Y 506.024,Z 342.437,A -85,B 0,C 180,E1 -5635.422,E2 -5635.422} C_VEL
LIN {X 0,Y 503.602,Z 343.472,A -85,B 0,C 180,E1 -5636.277,E2 -5636.277} C_VEL
LIN {X 0,Y 502.542,Z 344.18,A -85,B 0,C 180,E1 -5636.939,E2 -5636.939} C_VEL
LIN {X 0,Y 502.444,Z 344.392,A -85,B 0,C 180,E1 -5637.164,E2 -5637.164} C_VEL
LIN {X 0,Y 502.36,Z 347.18,A -85,B 0,C 180,E1 -5640.156,E2 -5640.156} C_VEL
LIN {X 0,Y 502.3,Z 349.394,A -85,B 0,C 180,E1 -5642.501,E2 -5642.501} C_VEL
LIN {X 0,Y 502.245,Z 352.34,A -85,B 0,C 180,E1 -5645.444,E2 -5645.444} C_VEL
LIN {X 0,Y 502.187,Z 355.723,A -85,B 0,C 180,E1 -5648.662,E2 -5648.662} C_VEL
LIN {X 0,Y 502.251,Z 357.282,A -85,B 0,C 180,E1 -5649.89,E2 -5649.89} C_VEL
LIN {X 0,Y 506.55,Z 371.981,A -85,B 0,C 180,E1 -5650.379,E2 -5650.379} C_VEL
LIN {X 0,Y 507.256,Z 376.124,A -85,B 0,C 180,E1 -5650.528,E2 -5650.528} C_VEL
LIN {X 0,Y 506.924,Z 390.567,A -85,B 0,C 180,E1 -5651.02,E2 -5651.02} C_VEL
LIN {X 0,Y 506.363,Z 405.477,A -85,B 0,C 180,E1 -5651.698,E2 -5651.698} C_VEL
LIN {X 0,Y 505.781,Z 419.447,A -85,B 0,C 180,E1 -5652.513,E2 -5652.513} C_VEL
LIN {X 0,Y 505.199,Z 432.206,A -85,B 0,C 180,E1 -5653.43,E2 -5653.43} C_VEL
LIN {X 0,Y 504.547,Z 444.337,A -85,B 0,C 180,E1 -5654.481,E2 -5654.481} C_VEL
LIN {X 0,Y 503.99,Z 455.756,A -85,B 0,C 180,E1 -5655.669,E2 -5655.669} C_VEL
LIN {X 0,Y 503.505,Z 465.658,A -85,B 0,C 180,E1 -5656.89,E2 -5656.89} C_VEL
LIN {X 0,Y 503.067,Z 475.32,A -85,B 0,C 180,E1 -5658.312,E2 -5658.312} C_VEL
LIN {X 0,Y 502.696,Z 483.37,A -85,B 0,C 180,E1 -5659.732,E2 -5659.732} C_VEL
LIN {X 0,Y 502.497,Z 490.002,A -85,B 0,C 180,E1 -5661.15,E2 -5661.15} C_VEL
LIN {X 0,Y 502.294,Z 496.148,A -85,B 0,C 180,E1 -5662.765,E2 -5662.765} C_VEL
LIN {X 0,Y 502.241,Z 500.89,A -85,B 0,C 180,E1 -5664.378,E2 -5664.378} C_VEL
LIN {X 0,Y 502.166,Z 504.369,A -85,B 0,C 180,E1 -5665.987,E2 -5665.987} C_VEL
LIN {X 0,Y 502.118,Z 506.672,A -85,B 0,C 180,E1 -5667.593,E2 -5667.593} C_VEL
LIN {X 0,Y 501.987,Z 507.857,A -85,B 0,C 180,E1 -5669.197,E2 -5669.197} C_VEL
LIN {X 0,Y 501.988,Z 507.876,A -85,B 0,C 180,E1 -5670.802,E2 -5670.802} C_VEL
LIN {X 0,Y 502.118,Z 506.765,A -85,B 0,C 180,E1 -5672.406,E2 -5672.406} C_VEL
LIN {X 0,Y 502.166,Z 504.535,A -85,B 0,C 180,E1 -5674.012,E2 -5674.012} C_VEL
LIN {X 0,Y 502.233,Z 501.126,A -85,B 0,C 180,E1 -5675.621,E2 -5675.621} C_VEL
LIN {X 0,Y 502.293,Z 496.459,A -85,B 0,C 180,E1 -5677.234,E2 -5677.234} C_VEL
LIN {X 0,Y 502.493,Z 490.404,A -85,B 0,C 180,E1 -5678.85,E2 -5678.85} C_VEL
LIN {X 0,Y 502.746,Z 482.778,A -85,B 0,C 180,E1 -5680.47,E2 -5680.47} C_VEL
LIN {X 0,Y 503.057,Z 474.697,A -85,B 0,C 180,E1 -5681.883,E2 -5681.883} C_VEL
LIN {X 0,Y 503.574,Z 464.831,A -85,B 0,C 180,E1 -5683.313,E2 -5683.313} C_VEL
LIN {X 0,Y 504.049,Z 454.767,A -85,B 0,C 180,E1 -5684.535,E2 -5684.535} C_VEL
LIN {X 0,Y 504.576,Z 443.722,A -85,B 0,C 180,E1 -5685.667,E2 -5685.667} C_VEL
LIN {X 0,Y 505.22,Z 432.03,A -85,B 0,C 180,E1 -5686.673,E2 -5686.673} C_VEL
LIN {X 0,Y 505.809,Z 419.246,A -85,B 0,C 180,E1 -5687.59,E2 -5687.59} C_VEL
LIN {X 0,Y 506.37,Z 405.218,A -85,B 0,C 180,E1 -5688.406,E2 -5688.406} C_VEL
LIN {X 0,Y 506.901,Z 391.098,A -85,B 0,C 180,E1 -5689.048,E2 -5689.048} C_VEL
LIN {X 0,Y 507.292,Z 376.219,A -85,B 0,C 180,E1 -5689.557,E2 -5689.557} C_VEL
LIN {X 0,Y 505.612,Z 368.352,A -85,B 0,C 180,E1 -5689.837,E2 -5689.837} C_VEL
LIN {X 0,Y 502.221,Z 356.978,A -85,B 0,C 180,E1 -5690.226,E2 -5690.226} C_VEL
LIN {X 0,Y 502.218,Z 353.968,A -85,B 0,C 180,E1 -5693.068,E2 -5693.068} C_VEL
LIN {X 0,Y 502.284,Z 351.257,A -85,B 0,C 180,E1 -5695.706,E2 -5695.706} C_VEL
LIN {X 0,Y 502.316,Z 348.632,A -85,B 0,C 180,E1 -5698.405,E2 -5698.405} C_VEL
LIN {X 0,Y 502.419,Z 345.787,A -85,B 0,C 180,E1 -5701.429,E2 -5701.429} C_VEL
LIN {X 0,Y 502.483,Z 343.047,A -85,B 0,C 180,E1 -5704.39,E2 -5704.39} C_VEL
LIN {X 0,Y 502.517,Z 340.54,A -85,B 0,C 180,E1 -5707.138,E2 -5707.138} C_VEL
LIN {X 0,Y 502.53,Z 338.876,A -85,B 0,C 180,E1 -5709.001,E2 -5709.001} C_VEL
LIN {X 0,Y 502.599,Z 338.507,A -85,B 0,C 180,E1 -5710.033,E2 -5710.033} C_VEL
LIN {X 0,Y 502.769,Z 338.48,A -85,B 0,C 180,E1 -5712.195,E2 -5712.195} C_VEL
LIN {X 0,Y 502.8,Z 338.478,A -85,B 0,C 180,E1 -5715.468,E2 -5715.468} C_VEL
LIN {X 0,Y 502.819,Z 338.479,A -85,B 0,C 180,E1 -5718.934,E2 -5718.934} C_VEL
LIN {X 0,Y 502.794,Z 338.482,A -85,B 0,C 180,E1 -5722.046,E2 -5722.046} C_VEL
LIN {X 0,Y 502.809,Z 338.48,A -85,B 0,C 180,E1 -5725.035,E2 -5725.035} C_VEL
LIN {X 0,Y 502.785,Z 338.477,A -85,B 0,C 180,E1 -5727.915,E2 -5727.915} C_VEL
LIN {X 0,Y 502.838,Z 338.473,A -85,B 0,C 180,E1 -5730.713,E2 -5730.713} C_VEL
LIN {X 0,Y 502.88,Z 338.463,A -85,B 0,C 180,E1 -5733.435,E2 -5733.435} C_VEL
LIN {X 0,Y 502.791,Z 338.482,A -85,B 0,C 180,E1 -5736.086,E2 -5736.086} C_VEL
LIN {X 0,Y 502.782,Z 338.479,A -85,B 0,C 180,E1 -5738.689,E2 -5738.689} C_VEL
LIN {X 0,Y 502.829,Z 338.471,A -85,B 0,C 180,E1 -5741.248,E2 -5741.248} C_VEL
LIN {X 0,Y 502.823,Z 338.476,A -85,B 0,C 180,E1 -5743.767,E2 -5743.767} C_VEL
LIN {X 0,Y 502.83,Z 338.471,A -85,B 0,C 180,E1 -5746.255,E2 -5746.255} C_VEL
LIN {X 0,Y 502.891,Z 338.464,A -85,B 0,C 180,E1 -5748.717,E2 -5748.717} C_VEL
LIN {X 0,Y 502.9,Z 338.465,A -85,B 0,C 180,E1 -5751.967,E2 -5751.967} C_VEL
LIN {X 0,Y 502.938,Z 338.463,A -85,B 0,C 180,E1 -5754.386,E2 -5754.386} C_VEL
LIN {X 0,Y 503.023,Z 338.452,A -85,B 0,C 180,E1 -5757.598,E2 -5757.598} C_VEL
LIN {X 0,Y 503.025,Z 338.453,A -85,B 0,C 180,E1 -5760,E2 -5760} C_VEL
LIN {X 0,Y 503.024,Z 338.45,A -85,B 0,C 180,E1 -5762.402,E2 -5762.402} C_VEL
LIN {X 0,Y 502.938,Z 338.461,A -85,B 0,C 180,E1 -5765.613,E2 -5765.613} C_VEL
LIN {X 0,Y 502.9,Z 338.469,A -85,B 0,C 180,E1 -5768.033,E2 -5768.033} C_VEL
LIN {X 0,Y 502.88,Z 338.469,A -85,B 0,C 180,E1 -5771.283,E2 -5771.283} C_VEL
LIN {X 0,Y 502.844,Z 338.472,A -85,B 0,C 180,E1 -5774.571,E2 -5774.571} C_VEL
LIN {X 0,Y 502.86,Z 338.47,A -85,B 0,C 180,E1 -5777.907,E2 -5777.907} C_VEL
LIN {X 0,Y 502.826,Z 338.475,A -85,B 0,C 180,E1 -5780.536,E2 -5780.536} C_VEL
LIN {X 0,Y 502.795,Z 338.484,A -85,B 0,C 180,E1 -5783.04,E2 -5783.04} C_VEL
LIN {X 0,Y 502.838,Z 338.475,A -85,B 0,C 180,E1 -5785.676,E2 -5785.676} C_VEL
LIN {X 0,Y 502.839,Z 338.474,A -85,B 0,C 180,E1 -5788.373,E2 -5788.373} C_VEL
LIN {X 0,Y 502.795,Z 338.479,A -85,B 0,C 180,E1 -5791.5,E2 -5791.5} C_VEL
LIN {X 0,Y 502.804,Z 338.479,A -85,B 0,C 180,E1 -5794.445,E2 -5794.445} C_VEL
LIN {X 0,Y 502.779,Z 338.483,A -85,B 0,C 180,E1 -5797.179,E2 -5797.179} C_VEL
LIN {X 0,Y 502.786,Z 338.483,A -85,B 0,C 180,E1 -5800.015,E2 -5800.015} C_VEL
LIN {X 0,Y 502.8,Z 338.48,A -85,B 0,C 180,E1 -5802.199,E2 -5802.199} C_VEL
LIN {X 0,Y 502.828,Z 338.627,A -85,B 0,C 180,E1 -5804.464,E2 -5804.464} C_VEL
LIN {X 0,Y 503.59,Z 343.205,A -85,B 0,C 180,E1 -5806.857,E2 -5806.857} C_VEL
LIN {X 0,Y 504.046,Z 347.282,A -85,B 0,C 180,E1 -5808.845,E2 -5808.845} C_VEL
LIN {X 0,Y 503.858,Z 352.876,A -85,B 0,C 180,E1 -5811.362,E2 -5811.362} C_VEL
LIN {X 0,Y 503.635,Z 359.294,A -85,B 0,C 180,E1 -5814.12,E2 -5814.12} C_VEL
LIN {X 0,Y 503.405,Z 366.371,A -85,B 0,C 180,E1 -5817.012,E2 -5817.012} C_VEL
LIN {X 0,Y 503.194,Z 373.514,A -85,B 0,C 180,E1 -5819.815,E2 -5819.815} C_VEL
LIN {X 0,Y 503.044,Z 379.467,A -85,B 0,C 180,E1 -5822.099,E2 -5822.099} C_VEL
LIN {X 0,Y 502.848,Z 387.726,A -85,B 0,C 180,E1 -5825.211,E2 -5825.211} C_VEL
LIN {X 0,Y 502.641,Z 397.048,A -85,B 0,C 180,E1 -5828.683,E2 -5828.683} C_VEL
LIN {X 0,Y 502.597,Z 400.094,A -85,B 0,C 180,E1 -5829.805,E2 -5829.805} C_VEL
LIN {X 0,Y 506.117,Z 415.761,A -85,B 0,C 180,E1 -5830.246,E2 -5830.246} C_VEL
LIN {X 0,Y 507.203,Z 421.184,A -85,B 0,C 180,E1 -5830.43,E2 -5830.43} C_VEL
LIN {X 0,Y 506.757,Z 435.321,A -85,B 0,C 180,E1 -5830.88,E2 -5830.88} C_VEL
LIN {X 0,Y 506.291,Z 449.462,A -85,B 0,C 180,E1 -5831.486,E2 -5831.486} C_VEL
LIN {X 0,Y 505.718,Z 462.601,A -85,B 0,C 180,E1 -5832.198,E2 -5832.198} C_VEL
LIN {X 0,Y 505.108,Z 476.267,A -85,B 0,C 180,E1 -5833.115,E2 -5833.115} C_VEL
LIN {X 0,Y 504.488,Z 489.841,A -85,B 0,C 180,E1 -5834.23,E2 -5834.23} C_VEL
LIN {X 0,Y 503.834,Z 502.201,A -85,B 0,C 180,E1 -5835.459,E2 -5835.459} C_VEL
LIN {X 0,Y 503.396,Z 512.517,A -85,B 0,C 180,E1 -5836.682,E2 -5836.682} C_VEL
LIN {X 0,Y 502.894,Z 523.056,A -85,B 0,C 180,E1 -5838.175,E2 -5838.175} C_VEL
LIN {X 0,Y 502.679,Z 530.994,A -85,B 0,C 180,E1 -5839.528,E2 -5839.528} C_VEL
LIN {X 0,Y 502.394,Z 538.873,A -85,B 0,C 180,E1 -5841.149,E2 -5841.149} C_VEL
LIN {X 0,Y 502.243,Z 545.146,A -85,B 0,C 180,E1 -5842.765,E2 -5842.765} C_VEL
LIN {X 0,Y 502.195,Z 550.002,A -85,B 0,C 180,E1 -5844.379,E2 -5844.379} C_VEL
LIN {X 0,Y 502.097,Z 553.556,A -85,B 0,C 180,E1 -5845.987,E2 -5845.987} C_VEL
LIN {X 0,Y 502.062,Z 555.896,A -85,B 0,C 180,E1 -5847.594,E2 -5847.594} C_VEL
LIN {X 0,Y 501.988,Z 557.07,A -85,B 0,C 180,E1 -5849.198,E2 -5849.198} C_VEL
LIN {X 0,Y 501.988,Z 557.069,A -85,B 0,C 180,E1 -5850.803,E2 -5850.803} C_VEL
LIN {X 0,Y 502.062,Z 555.891,A -85,B 0,C 180,E1 -5852.407,E2 -5852.407} C_VEL
LIN {X 0,Y 502.097,Z 553.55,A -85,B 0,C 180,E1 -5854.014,E2 -5854.014} C_VEL
LIN {X 0,Y 502.197,Z 550.001,A -85,B 0,C 180,E1 -5855.622,E2 -5855.622} C_VEL
LIN {X 0,Y 502.246,Z 545.148,A -85,B 0,C 180,E1 -5857.235,E2 -5857.235} C_VEL
LIN {X 0,Y 502.394,Z 538.866,A -85,B 0,C 180,E1 -5858.852,E2 -5858.852} C_VEL
LIN {X 0,Y 502.679,Z 530.984,A -85,B 0,C 180,E1 -5860.472,E2 -5860.472} C_VEL
LIN {X 0,Y 502.925,Z 522.949,A -85,B 0,C 180,E1 -5861.841,E2 -5861.841} C_VEL
LIN {X 0,Y 503.397,Z 512.512,A -85,B 0,C 180,E1 -5863.319,E2 -5863.319} C_VEL
LIN {X 0,Y 503.824,Z 502.196,A -85,B 0,C 180,E1 -5864.542,E2 -5864.542} C_VEL
LIN {X 0,Y 504.445,Z 489.773,A -85,B 0,C 180,E1 -5865.778,E2 -5865.778} C_VEL
LIN {X 0,Y 505.095,Z 476.263,A -85,B 0,C 180,E1 -5866.886,E2 -5866.886} C_VEL
LIN {X 0,Y 505.741,Z 462.582,A -85,B 0,C 180,E1 -5867.802,E2 -5867.802} C_VEL
LIN {X 0,Y 506.351,Z 448.423,A -85,B 0,C 180,E1 -5868.564,E2 -5868.564} C_VEL
LIN {X 0,Y 506.839,Z 433.308,A -85,B 0,C 180,E1 -5869.196,E2 -5869.196} C_VEL
LIN {X 0,Y 507.037,Z 419.773,A -85,B 0,C 180,E1 -5869.617,E2 -5869.617} C_VEL
LIN {X 0,Y 503.555,Z 404.737,A -85,B 0,C 180,E1 -5870.08,E2 -5870.08} C_VEL
LIN {X 0,Y 502.574,Z 400.073,A -85,B 0,C 180,E1 -5870.203,E2 -5870.203} C_VEL
LIN {X 0,Y 502.699,Z 392.381,A -85,B 0,C 180,E1 -5873.045,E2 -5873.045} C_VEL
LIN {X 0,Y 502.959,Z 384.187,A -85,B 0,C 180,E1 -5876.114,E2 -5876.114} C_VEL
LIN {X 0,Y 503.175,Z 375.841,A -85,B 0,C 180,E1 -5879.266,E2 -5879.266} C_VEL
LIN {X 0,Y 503.349,Z 367.507,A -85,B 0,C 180,E1 -5882.518,E2 -5882.518} C_VEL
LIN {X 0,Y 503.605,Z 360.444,A -85,B 0,C 180,E1 -5885.391,E2 -5885.391} C_VEL
LIN {X 0,Y 503.791,Z 354.588,A -85,B 0,C 180,E1 -5887.866,E2 -5887.866} C_VEL
LIN {X 0,Y 503.969,Z 348.82,A -85,B 0,C 180,E1 -5890.425,E2 -5890.425} C_VEL
LIN {X 0,Y 503.844,Z 344.802,A -85,B 0,C 180,E1 -5892.33,E2 -5892.33} C_VEL
LIN {X 0,Y 503.168,Z 340.402,A -85,B 0,C 180,E1 -5894.574,E2 -5894.574} C_VEL
LIN {X 0,Y 502.788,Z 338.477,A -85,B 0,C 180,E1 -5895.661,E2 -5895.661} C_VEL
LIN {X 0,Y 502.82,Z 338.478,A -85,B 0,C 180,E1 -5899.005,E2 -5899.005} C_VEL
LIN {X 0,Y 502.797,Z 338.484,A -85,B 0,C 180,E1 -5902.046,E2 -5902.046} C_VEL
LIN {X 0,Y 502.812,Z 338.481,A -85,B 0,C 180,E1 -5905.035,E2 -5905.035} C_VEL
LIN {X 0,Y 502.785,Z 338.484,A -85,B 0,C 180,E1 -5907.916,E2 -5907.916} C_VEL
LIN {X 0,Y 502.827,Z 338.479,A -85,B 0,C 180,E1 -5910.712,E2 -5910.712} C_VEL
LIN {X 0,Y 502.865,Z 338.471,A -85,B 0,C 180,E1 -5913.439,E2 -5913.439} C_VEL
LIN {X 0,Y 502.787,Z 338.48,A -85,B 0,C 180,E1 -5916.086,E2 -5916.086} C_VEL
LIN {X 0,Y 502.787,Z 338.483,A -85,B 0,C 180,E1 -5918.689,E2 -5918.689} C_VEL
LIN {X 0,Y 502.833,Z 338.476,A -85,B 0,C 180,E1 -5921.248,E2 -5921.248} C_VEL
LIN {X 0,Y 502.826,Z 338.476,A -85,B 0,C 180,E1 -5923.767,E2 -5923.767} C_VEL
LIN {X 0,Y 502.835,Z 338.479,A -85,B 0,C 180,E1 -5926.255,E2 -5926.255} C_VEL
LIN {X 0,Y 502.881,Z 338.47,A -85,B 0,C 180,E1 -5928.717,E2 -5928.717} C_VEL
LIN {X 0,Y 502.905,Z 338.468,A -85,B 0,C 180,E1 -5931.967,E2 -5931.967} C_VEL
LIN {X 0,Y 502.941,Z 338.461,A -85,B 0,C 180,E1 -5934.387,E2 -5934.387} C_VEL
LIN {X 0,Y 503.028,Z 338.449,A -85,B 0,C 180,E1 -5937.598,E2 -5937.598} C_VEL
LIN {X 0,Y 503.03,Z 338.452,A -85,B 0,C 180,E1 -5940,E2 -5940} C_VEL
LIN {X 0,Y 503.027,Z 338.45,A -85,B 0,C 180,E1 -5942.402,E2 -5942.402} C_VEL
LIN {X 0,Y 502.943,Z 338.462,A -85,B 0,C 180,E1 -5945.614,E2 -5945.614} C_VEL
LIN {X 0,Y 502.906,Z 338.465,A -85,B 0,C 180,E1 -5948.033,E2 -5948.033} C_VEL
LIN {X 0,Y 502.881,Z 338.464,A -85,B 0,C 180,E1 -5951.283,E2 -5951.283} C_VEL
LIN {X 0,Y 502.849,Z 338.468,A -85,B 0,C 180,E1 -5954.571,E2 -5954.571} C_VEL
LIN {X 0,Y 502.866,Z 338.472,A -85,B 0,C 180,E1 -5957.907,E2 -5957.907} C_VEL
LIN {X 0,Y 502.832,Z 338.464,A -85,B 0,C 180,E1 -5960.536,E2 -5960.536} C_VEL
LIN {X 0,Y 502.791,Z 338.48,A -85,B 0,C 180,E1 -5963.041,E2 -5963.041} C_VEL
LIN {X 0,Y 502.825,Z 338.476,A -85,B 0,C 180,E1 -5965.676,E2 -5965.676} C_VEL
LIN {X 0,Y 502.843,Z 338.469,A -85,B 0,C 180,E1 -5968.373,E2 -5968.373} C_VEL
LIN {X 0,Y 502.796,Z 338.48,A -85,B 0,C 180,E1 -5971.499,E2 -5971.499} C_VEL
LIN {X 0,Y 502.808,Z 338.474,A -85,B 0,C 180,E1 -5974.444,E2 -5974.444} C_VEL
LIN {X 0,Y 502.785,Z 338.48,A -85,B 0,C 180,E1 -5977.178,E2 -5977.178} C_VEL
LIN {X 0,Y 502.791,Z 338.48,A -85,B 0,C 180,E1 -5980.015,E2 -5980.015} C_VEL
LIN {X 0,Y 502.806,Z 338.48,A -85,B 0,C 180,E1 -5982.199,E2 -5982.199} C_VEL
LIN {X 0,Y 502.804,Z 338.484,A -85,B 0,C 180,E1 -5985.468,E2 -5985.468} C_VEL
LIN {X 0,Y 502.767,Z 338.484,A -85,B 0,C 180,E1 -5987.857,E2 -5987.857} C_VEL
LIN {X 0,Y 502.574,Z 338.511,A -85,B 0,C 180,E1 -5990.275,E2 -5990.275} C_VEL
LIN {X 0,Y 502.5,Z 339.289,A -85,B 0,C 180,E1 -5991.556,E2 -5991.556} C_VEL
LIN {X 0,Y 502.489,Z 341.681,A -85,B 0,C 180,E1 -5994.215,E2 -5994.215} C_VEL
LIN {X 0,Y 502.444,Z 344.392,A -85,B 0,C 180,E1 -5997.164,E2 -5997.164} C_VEL
LIN {X 0,Y 501.739,Z 345.066,A -85,B 0,C 180,E1 -5997.828,E2 -5997.828} C_VEL
LIN {X 0,Y 498.843,Z 346.35,A -85,B 0,C 180,E1 -5998.904,E2 -5998.904} C_VEL
LIN {X 0,Y 496.406,Z 347.4,A -85,B 0,C 180,E1 -5999.771,E2 -5999.771} C_VEL
LIN {X 0,Y 495.351,Z 348.12,A -85,B 0,C 180,E1 -6000.442,E2 -6000.442} C_VEL
LIN {X 0,Y 495.259,Z 348.338,A -85,B 0,C 180,E1 -6000.67,E2 -6000.67} C_VEL
LIN {X 0,Y 495.237,Z 350.918,A -85,B 0,C 180,E1 -6003.386,E2 -6003.386} C_VEL
LIN {X 0,Y 495.158,Z 354.141,A -85,B 0,C 180,E1 -6006.583,E2 -6006.583} C_VEL
LIN {X 0,Y 495.137,Z 357.362,A -85,B 0,C 180,E1 -6009.582,E2 -6009.582} C_VEL
LIN {X 0,Y 499.777,Z 373.027,A -85,B 0,C 180,E1 -6010.122,E2 -6010.122} C_VEL
LIN {X 0,Y 500.56,Z 377.585,A -85,B 0,C 180,E1 -6010.289,E2 -6010.289} C_VEL
LIN {X 0,Y 500.199,Z 392.447,A -85,B 0,C 180,E1 -6010.818,E2 -6010.818} C_VEL
LIN {X 0,Y 499.629,Z 405.837,A -85,B 0,C 180,E1 -6011.442,E2 -6011.442} C_VEL
LIN {X 0,Y 499.024,Z 419.804,A -85,B 0,C 180,E1 -6012.268,E2 -6012.268} C_VEL
LIN {X 0,Y 498.387,Z 432.558,A -85,B 0,C 180,E1 -6013.197,E2 -6013.197} C_VEL
LIN {X 0,Y 497.702,Z 444.804,A -85,B 0,C 180,E1 -6014.273,E2 -6014.273} C_VEL
LIN {X 0,Y 497.085,Z 456.111,A -85,B 0,C 180,E1 -6015.466,E2 -6015.466} C_VEL
LIN {X 0,Y 496.569,Z 466.012,A -85,B 0,C 180,E1 -6016.703,E2 -6016.703} C_VEL
LIN {X 0,Y 496.124,Z 474.682,A -85,B 0,C 180,E1 -6017.981,E2 -6017.981} C_VEL
LIN {X 0,Y 495.749,Z 482.634,A -85,B 0,C 180,E1 -6019.38,E2 -6019.38} C_VEL
LIN {X 0,Y 495.462,Z 490.354,A -85,B 0,C 180,E1 -6021.023,E2 -6021.023} C_VEL
LIN {X 0,Y 495.236,Z 496.499,A -85,B 0,C 180,E1 -6022.662,E2 -6022.662} C_VEL
LIN {X 0,Y 495.18,Z 501.24,A -85,B 0,C 180,E1 -6024.298,E2 -6024.298} C_VEL
LIN {X 0,Y 495.099,Z 504.717,A -85,B 0,C 180,E1 -6025.93,E2 -6025.93} C_VEL
LIN {X 0,Y 495.05,Z 507.019,A -85,B 0,C 180,E1 -6027.559,E2 -6027.559} C_VEL
LIN {X 0,Y 494.907,Z 508.204,A -85,B 0,C 180,E1 -6029.186,E2 -6029.186} C_VEL
LIN {X 0,Y 494.908,Z 508.222,A -85,B 0,C 180,E1 -6030.813,E2 -6030.813} C_VEL
LIN {X 0,Y 495.051,Z 507.111,A -85,B 0,C 180,E1 -6032.441,E2 -6032.441} C_VEL
LIN {X 0,Y 495.099,Z 504.881,A -85,B 0,C 180,E1 -6034.07,E2 -6034.07} C_VEL
LIN {X 0,Y 495.165,Z 501.472,A -85,B 0,C 180,E1 -6035.702,E2 -6035.702} C_VEL
LIN {X 0,Y 495.235,Z 496.805,A -85,B 0,C 180,E1 -6037.338,E2 -6037.338} C_VEL
LIN {X 0,Y 495.455,Z 490.751,A -85,B 0,C 180,E1 -6038.976,E2 -6038.976} C_VEL
LIN {X 0,Y 495.743,Z 483.124,A -85,B 0,C 180,E1 -6040.62,E2 -6040.62} C_VEL
LIN {X 0,Y 496.131,Z 474.116,A -85,B 0,C 180,E1 -6042.197,E2 -6042.197} C_VEL
LIN {X 0,Y 496.645,Z 465.175,A -85,B 0,C 180,E1 -6043.502,E2 -6043.502} C_VEL
LIN {X 0,Y 497.174,Z 455.11,A -85,B 0,C 180,E1 -6044.74,E2 -6044.74} C_VEL
LIN {X 0,Y 497.715,Z 444.307,A -85,B 0,C 180,E1 -6045.865,E2 -6045.865} C_VEL
LIN {X 0,Y 498.413,Z 432.371,A -85,B 0,C 180,E1 -6046.907,E2 -6046.907} C_VEL
LIN {X 0,Y 499.053,Z 419.583,A -85,B 0,C 180,E1 -6047.836,E2 -6047.836} C_VEL
LIN {X 0,Y 499.638,Z 405.553,A -85,B 0,C 180,E1 -6048.663,E2 -6048.663} C_VEL
LIN {X 0,Y 500.209,Z 390.555,A -85,B 0,C 180,E1 -6049.349,E2 -6049.349} C_VEL
LIN {X 0,Y 500.488,Z 376.187,A -85,B 0,C 180,E1 -6049.845,E2 -6049.845} C_VEL
LIN {X 0,Y 497.269,Z 364.306,A -85,B 0,C 180,E1 -6050.288,E2 -6050.288} C_VEL
LIN {X 0,Y 495.113,Z 357.3,A -85,B 0,C 180,E1 -6050.512,E2 -6050.512} C_VEL
LIN {X 0,Y 495.16,Z 354.241,A -85,B 0,C 180,E1 -6053.416,E2 -6053.416} C_VEL
LIN {X 0,Y 495.235,Z 351.009,A -85,B 0,C 180,E1 -6056.613,E2 -6056.613} C_VEL
LIN {X 0,Y 495.292,Z 348.028,A -85,B 0,C 180,E1 -6059.777,E2 -6059.777} C_VEL
LIN {X 0,Y 495.368,Z 345.407,A -85,B 0,C 180,E1 -6062.623,E2 -6062.623} C_VEL
LIN {X 0,Y 495.41,Z 342.714,A -85,B 0,C 180,E1 -6065.565,E2 -6065.565} C_VEL
LIN {X 0,Y 495.461,Z 340.888,A -85,B 0,C 180,E1 -6067.585,E2 -6067.585} C_VEL
LIN {X 0,Y 495.496,Z 339.392,A -85,B 0,C 180,E1 -6069.662,E2 -6069.662} C_VEL
LIN {X 0,Y 495.716,Z 339.359,A -85,B 0,C 180,E1 -6072.504,E2 -6072.504} C_VEL
LIN {X 0,Y 495.748,Z 339.357,A -85,B 0,C 180,E1 -6075.139,E2 -6075.139} C_VEL
LIN {X 0,Y 495.757,Z 339.356,A -85,B 0,C 180,E1 -6078.219,E2 -6078.219} C_VEL
LIN {X 0,Y 495.75,Z 339.356,A -85,B 0,C 180,E1 -6081.408,E2 -6081.408} C_VEL
LIN {X 0,Y 495.757,Z 339.355,A -85,B 0,C 180,E1 -6084.463,E2 -6084.463} C_VEL
LIN {X 0,Y 495.767,Z 339.35,A -85,B 0,C 180,E1 -6087.406,E2 -6087.406} C_VEL
LIN {X 0,Y 495.781,Z 339.353,A -85,B 0,C 180,E1 -6090.254,E2 -6090.254} C_VEL
LIN {X 0,Y 495.833,Z 339.342,A -85,B 0,C 180,E1 -6093.248,E2 -6093.248} C_VEL
LIN {X 0,Y 495.752,Z 339.358,A -85,B 0,C 180,E1 -6095.725,E2 -6095.725} C_VEL
LIN {X 0,Y 495.746,Z 339.353,A -85,B 0,C 180,E1 -6098.371,E2 -6098.371} C_VEL
LIN {X 0,Y 495.784,Z 339.349,A -85,B 0,C 180,E1 -6100.971,E2 -6100.971} C_VEL
LIN {X 0,Y 495.78,Z 339.356,A -85,B 0,C 180,E1 -6103.53,E2 -6103.53} C_VEL
LIN {X 0,Y 495.793,Z 339.346,A -85,B 0,C 180,E1 -6106.056,E2 -6106.056} C_VEL
LIN {X 0,Y 495.866,Z 339.34,A -85,B 0,C 180,E1 -6108.555,E2 -6108.555} C_VEL
LIN {X 0,Y 495.872,Z 339.34,A -85,B 0,C 180,E1 -6111.852,E2 -6111.852} C_VEL
LIN {X 0,Y 495.896,Z 339.342,A -85,B 0,C 180,E1 -6114.306,E2 -6114.306} C_VEL
LIN {X 0,Y 495.992,Z 339.328,A -85,B 0,C 180,E1 -6117.564,E2 -6117.564} C_VEL
LIN {X 0,Y 495.996,Z 339.329,A -85,B 0,C 180,E1 -6120,E2 -6120} C_VEL
LIN {X 0,Y 495.992,Z 339.326,A -85,B 0,C 180,E1 -6122.436,E2 -6122.436} C_VEL
LIN {X 0,Y 495.895,Z 339.339,A -85,B 0,C 180,E1 -6125.693,E2 -6125.693} C_VEL
LIN {X 0,Y 495.871,Z 339.343,A -85,B 0,C 180,E1 -6128.148,E2 -6128.148} C_VEL
LIN {X 0,Y 495.853,Z 339.343,A -85,B 0,C 180,E1 -6131.445,E2 -6131.445} C_VEL
LIN {X 0,Y 495.788,Z 339.351,A -85,B 0,C 180,E1 -6134.783,E2 -6134.783} C_VEL
LIN {X 0,Y 495.785,Z 339.353,A -85,B 0,C 180,E1 -6137.319,E2 -6137.319} C_VEL
LIN {X 0,Y 495.776,Z 339.357,A -85,B 0,C 180,E1 -6139.89,E2 -6139.89} C_VEL
LIN {X 0,Y 495.756,Z 339.359,A -85,B 0,C 180,E1 -6142.86,E2 -6142.86} C_VEL
LIN {X 0,Y 495.789,Z 339.357,A -85,B 0,C 180,E1 -6146.068,E2 -6146.068} C_VEL
LIN {X 0,Y 495.777,Z 339.356,A -85,B 0,C 180,E1 -6148.814,E2 -6148.814} C_VEL
LIN {X 0,Y 495.757,Z 339.357,A -85,B 0,C 180,E1 -6151.726,E2 -6151.726} C_VEL
LIN {X 0,Y 495.774,Z 339.355,A -85,B 0,C 180,E1 -6154.695,E2 -6154.695} C_VEL
LIN {X 0,Y 495.73,Z 339.36,A -85,B 0,C 180,E1 -6157.562,E2 -6157.562} C_VEL
LIN {X 0,Y 495.765,Z 339.357,A -85,B 0,C 180,E1 -6160.7,E2 -6160.7} C_VEL
LIN {X 0,Y 495.732,Z 339.359,A -85,B 0,C 180,E1 -6164.001,E2 -6164.001} C_VEL
LIN {X 0,Y 496.44,Z 343.391,A -85,B 0,C 180,E1 -6166.219,E2 -6166.219} C_VEL
LIN {X 0,Y 497.035,Z 348.007,A -85,B 0,C 180,E1 -6168.539,E2 -6168.539} C_VEL
LIN {X 0,Y 496.975,Z 352.189,A -85,B 0,C 180,E1 -6170.479,E2 -6170.479} C_VEL
LIN {X 0,Y 496.696,Z 359.625,A -85,B 0,C 180,E1 -6173.757,E2 -6173.757} C_VEL
LIN {X 0,Y 496.404,Z 366.57,A -85,B 0,C 180,E1 -6176.648,E2 -6176.648} C_VEL
LIN {X 0,Y 496.194,Z 373.288,A -85,B 0,C 180,E1 -6179.343,E2 -6179.343} C_VEL
LIN {X 0,Y 495.988,Z 380.4,A -85,B 0,C 180,E1 -6182.122,E2 -6182.122} C_VEL
LIN {X 0,Y 495.799,Z 388.245,A -85,B 0,C 180,E1 -6185.122,E2 -6185.122} C_VEL
LIN {X 0,Y 495.58,Z 396.789,A -85,B 0,C 180,E1 -6188.364,E2 -6188.364} C_VEL
LIN {X 0,Y 495.528,Z 399.789,A -85,B 0,C 180,E1 -6189.501,E2 -6189.501} C_VEL
LIN {X 0,Y 499.38,Z 416.812,A -85,B 0,C 180,E1 -6190.001,E2 -6190.001} C_VEL
LIN {X 0,Y 500.478,Z 421.754,A -85,B 0,C 180,E1 -6190.183,E2 -6190.183} C_VEL
LIN {X 0,Y 500.002,Z 435.662,A -85,B 0,C 180,E1 -6190.64,E2 -6190.64} C_VEL
LIN {X 0,Y 499.504,Z 449.11,A -85,B 0,C 180,E1 -6191.226,E2 -6191.226} C_VEL
LIN {X 0,Y 498.908,Z 462.25,A -85,B 0,C 180,E1 -6191.947,E2 -6191.947} C_VEL
LIN {X 0,Y 498.251,Z 475.916,A -85,B 0,C 180,E1 -6192.876,E2 -6192.876} C_VEL
LIN {X 0,Y 497.596,Z 489.177,A -85,B 0,C 180,E1 -6193.977,E2 -6193.977} C_VEL
LIN {X 0,Y 496.881,Z 501.849,A -85,B 0,C 180,E1 -6195.251,E2 -6195.251} C_VEL
LIN {X 0,Y 496.41,Z 512.165,A -85,B 0,C 180,E1 -6196.491,E2 -6196.491} C_VEL
LIN {X 0,Y 495.877,Z 522.289,A -85,B 0,C 180,E1 -6197.939,E2 -6197.939} C_VEL
LIN {X 0,Y 495.644,Z 530.643,A -85,B 0,C 180,E1 -6199.378,E2 -6199.378} C_VEL
LIN {X 0,Y 495.32,Z 538.522,A -85,B 0,C 180,E1 -6201.021,E2 -6201.021} C_VEL
LIN {X 0,Y 495.164,Z 544.797,A -85,B 0,C 180,E1 -6202.661,E2 -6202.661} C_VEL
LIN {X 0,Y 495.106,Z 549.653,A -85,B 0,C 180,E1 -6204.298,E2 -6204.298} C_VEL
LIN {X 0,Y 494.996,Z 553.207,A -85,B 0,C 180,E1 -6205.929,E2 -6205.929} C_VEL
LIN {X 0,Y 494.971,Z 555.548,A -85,B 0,C 180,E1 -6207.559,E2 -6207.559} C_VEL
LIN {X 0,Y 494.908,Z 556.723,A -85,B 0,C 180,E1 -6209.187,E2 -6209.187} C_VEL
LIN {X 0,Y 494.908,Z 556.722,A -85,B 0,C 180,E1 -6210.814,E2 -6210.814} C_VEL
LIN {X 0,Y 494.971,Z 555.543,A -85,B 0,C 180,E1 -6212.442,E2 -6212.442} C_VEL
LIN {X 0,Y 494.996,Z 553.202,A -85,B 0,C 180,E1 -6214.071,E2 -6214.071} C_VEL
LIN {X 0,Y 495.11,Z 549.652,A -85,B 0,C 180,E1 -6215.703,E2 -6215.703} C_VEL
LIN {X 0,Y 495.166,Z 544.798,A -85,B 0,C 180,E1 -6217.339,E2 -6217.339} C_VEL
LIN {X 0,Y 495.32,Z 538.515,A -85,B 0,C 180,E1 -6218.98,E2 -6218.98} C_VEL
LIN {X 0,Y 495.644,Z 530.633,A -85,B 0,C 180,E1 -6220.623,E2 -6220.623} C_VEL
LIN {X 0,Y 495.891,Z 522.236,A -85,B 0,C 180,E1 -6222.068,E2 -6222.068} C_VEL
LIN {X 0,Y 496.411,Z 512.16,A -85,B 0,C 180,E1 -6223.509,E2 -6223.509} C_VEL
LIN {X 0,Y 496.859,Z 501.843,A -85,B 0,C 180,E1 -6224.751,E2 -6224.751} C_VEL
LIN {X 0,Y 497.509,Z 490.03,A -85,B 0,C 180,E1 -6225.945,E2 -6225.945} C_VEL
LIN {X 0,Y 498.162,Z 477.252,A -85,B 0,C 180,E1 -6227.022,E2 -6227.022} C_VEL
LIN {X 0,Y 498.848,Z 463.864,A -85,B 0,C 180,E1 -6227.95,E2 -6227.95} C_VEL
LIN {X 0,Y 499.458,Z 451.094,A -85,B 0,C 180,E1 -6228.671,E2 -6228.671} C_VEL
LIN {X 0,Y 499.952,Z 436.954,A -85,B 0,C 180,E1 -6229.31,E2 -6229.31} C_VEL
LIN {X 0,Y 500.399,Z 421.466,A -85,B 0,C 180,E1 -6229.829,E2 -6229.829} C_VEL
LIN {X 0,Y 496.748,Z 405.505,A -85,B 0,C 180,E1 -6230.347,E2 -6230.347} C_VEL
LIN {X 0,Y 495.526,Z 399.788,A -85,B 0,C 180,E1 -6230.498,E2 -6230.498} C_VEL
LIN {X 0,Y 495.661,Z 392.155,A -85,B 0,C 180,E1 -6233.392,E2 -6233.392} C_VEL
LIN {X 0,Y 495.889,Z 385.112,A -85,B 0,C 180,E1 -6236.063,E2 -6236.063} C_VEL
LIN {X 0,Y 496.138,Z 376.809,A -85,B 0,C 180,E1 -6239.256,E2 -6239.256} C_VEL
LIN {X 0,Y 496.328,Z 368.479,A -85,B 0,C 180,E1 -6242.553,E2 -6242.553} C_VEL
LIN {X 0,Y 496.598,Z 361.431,A -85,B 0,C 180,E1 -6245.468,E2 -6245.468} C_VEL
LIN {X 0,Y 496.833,Z 354.437,A -85,B 0,C 180,E1 -6248.492,E2 -6248.492} C_VEL
LIN {X 0,Y 497.016,Z 349.831,A -85,B 0,C 180,E1 -6250.577,E2 -6250.577} C_VEL
LIN {X 0,Y 496.775,Z 345.583,A -85,B 0,C 180,E1 -6252.637,E2 -6252.637} C_VEL
LIN {X 0,Y 495.898,Z 340.236,A -85,B 0,C 180,E1 -6255.45,E2 -6255.45} C_VEL
LIN {X 0,Y 495.734,Z 339.356,A -85,B 0,C 180,E1 -6255.999,E2 -6255.999} C_VEL
LIN {X 0,Y 495.768,Z 339.356,A -85,B 0,C 180,E1 -6259.3,E2 -6259.3} C_VEL
LIN {X 0,Y 495.734,Z 339.362,A -85,B 0,C 180,E1 -6262.439,E2 -6262.439} C_VEL
LIN {X 0,Y 495.788,Z 339.354,A -85,B 0,C 180,E1 -6265.458,E2 -6265.458} C_VEL
LIN {X 0,Y 495.757,Z 339.357,A -85,B 0,C 180,E1 -6268.364,E2 -6268.364} C_VEL
LIN {X 0,Y 495.791,Z 339.352,A -85,B 0,C 180,E1 -6271.507,E2 -6271.507} C_VEL
LIN {X 0,Y 495.794,Z 339.356,A -85,B 0,C 180,E1 -6273.932,E2 -6273.932} C_VEL
LIN {X 0,Y 495.762,Z 339.358,A -85,B 0,C 180,E1 -6277.14,E2 -6277.14} C_VEL
LIN {X 0,Y 495.775,Z 339.357,A -85,B 0,C 180,E1 -6280.11,E2 -6280.11} C_VEL
LIN {X 0,Y 495.79,Z 339.353,A -85,B 0,C 180,E1 -6282.682,E2 -6282.682} C_VEL
LIN {X 0,Y 495.794,Z 339.352,A -85,B 0,C 180,E1 -6285.217,E2 -6285.217} C_VEL
LIN {X 0,Y 495.855,Z 339.345,A -85,B 0,C 180,E1 -6288.555,E2 -6288.555} C_VEL
LIN {X 0,Y 495.876,Z 339.343,A -85,B 0,C 180,E1 -6291.852,E2 -6291.852} C_VEL
LIN {X 0,Y 495.899,Z 339.338,A -85,B 0,C 180,E1 -6294.307,E2 -6294.307} C_VEL
LIN {X 0,Y 495.997,Z 339.325,A -85,B 0,C 180,E1 -6297.564,E2 -6297.564} C_VEL
LIN {X 0,Y 496.009,Z 339.324,A -85,B 0,C 180,E1 -6300.812,E2 -6300.812} C_VEL
LIN {X 0,Y 495.846,Z 339.344,A -85,B 0,C 180,E1 -6303.25,E2 -6303.25} C_VEL
LIN {X 0,Y 495.884,Z 339.338,A -85,B 0,C 180,E1 -6306.51,E2 -6306.51} C_VEL
LIN {X 0,Y 495.847,Z 339.349,A -85,B 0,C 180,E1 -6308.97,E2 -6308.97} C_VEL
LIN {X 0,Y 495.832,Z 339.339,A -85,B 0,C 180,E1 -6312.035,E2 -6312.035} C_VEL
LIN {X 0,Y 495.828,Z 339.347,A -85,B 0,C 180,E1 -6315.452,E2 -6315.452} C_VEL
LIN {X 0,Y 495.81,Z 339.348,A -85,B 0,C 180,E1 -6318.247,E2 -6318.247} C_VEL
LIN {X 0,Y 495.778,Z 339.343,A -85,B 0,C 180,E1 -6320.756,E2 -6320.756} C_VEL
LIN {X 0,Y 495.746,Z 339.356,A -85,B 0,C 180,E1 -6323.387,E2 -6323.387} C_VEL
LIN {X 0,Y 495.827,Z 339.342,A -85,B 0,C 180,E1 -6326.749,E2 -6326.749} C_VEL
LIN {X 0,Y 495.77,Z 339.353,A -85,B 0,C 180,E1 -6329.746,E2 -6329.746} C_VEL
LIN {X 0,Y 495.771,Z 339.35,A -85,B 0,C 180,E1 -6332.594,E2 -6332.594} C_VEL
LIN {X 0,Y 495.759,Z 339.355,A -85,B 0,C 180,E1 -6335.537,E2 -6335.537} C_VEL
LIN {X 0,Y 495.767,Z 339.354,A -85,B 0,C 180,E1 -6338.768,E2 -6338.768} C_VEL
LIN {X 0,Y 495.76,Z 339.356,A -85,B 0,C 180,E1 -6341.781,E2 -6341.781} C_VEL
LIN {X 0,Y 495.753,Z 339.359,A -85,B 0,C 180,E1 -6345.139,E2 -6345.139} C_VEL
LIN {X 0,Y 495.705,Z 339.366,A -85,B 0,C 180,E1 -6348.213,E2 -6348.213} C_VEL
LIN {X 0,Y 495.518,Z 339.39,A -85,B 0,C 180,E1 -6350.339,E2 -6350.339} C_VEL
LIN {X 0,Y 495.447,Z 339.896,A -85,B 0,C 180,E1 -6351.38,E2 -6351.38} C_VEL
LIN {X 0,Y 495.43,Z 342.186,A -85,B 0,C 180,E1 -6353.958,E2 -6353.958} C_VEL
LIN {X 0,Y 495.383,Z 344.792,A -85,B 0,C 180,E1 -6356.828,E2 -6356.828} C_VEL
LIN {X 0,Y 495.312,Z 347.038,A -85,B 0,C 180,E1 -6359.282,E2 -6359.282} C_VEL
LIN {X 0,Y 495.259,Z 348.338,A -85,B 0,C 180,E1 -6360.67,E2 -6360.67} C_VEL
LIN {X 0,Y 494.571,Z 349.033,A -85,B 0,C 180,E1 -6361.344,E2 -6361.344} C_VEL
LIN {X 0,Y 491.687,Z 350.349,A -85,B 0,C 180,E1 -6362.435,E2 -6362.435} C_VEL
LIN {X 0,Y 489.262,Z 351.432,A -85,B 0,C 180,E1 -6363.315,E2 -6363.315} C_VEL
LIN {X 0,Y 488.228,Z 352.197,A -85,B 0,C 180,E1 -6363.995,E2 -6363.995} C_VEL
LIN {X 0,Y 488.148,Z 352.433,A -85,B 0,C 180,E1 -6364.226,E2 -6364.226} C_VEL
LIN {X 0,Y 488.083,Z 355.375,A -85,B 0,C 180,E1 -6367.154,E2 -6367.154} C_VEL
LIN {X 0,Y 488.072,Z 357.788,A -85,B 0,C 180,E1 -6369.274,E2 -6369.274} C_VEL
LIN {X 0,Y 492.808,Z 373.192,A -85,B 0,C 180,E1 -6369.822,E2 -6369.822} C_VEL
LIN {X 0,Y 493.89,Z 378.59,A -85,B 0,C 180,E1 -6370.03,E2 -6370.03} C_VEL
LIN {X 0,Y 493.499,Z 393.157,A -85,B 0,C 180,E1 -6370.561,E2 -6370.561} C_VEL
LIN {X 0,Y 492.926,Z 406.197,A -85,B 0,C 180,E1 -6371.181,E2 -6371.181} C_VEL
LIN {X 0,Y 492.284,Z 420.161,A -85,B 0,C 180,E1 -6372.017,E2 -6372.017} C_VEL
LIN {X 0,Y 491.58,Z 432.915,A -85,B 0,C 180,E1 -6372.957,E2 -6372.957} C_VEL
LIN {X 0,Y 490.864,Z 445.285,A -85,B 0,C 180,E1 -6374.061,E2 -6374.061} C_VEL
LIN {X 0,Y 490.2,Z 456.466,A -85,B 0,C 180,E1 -6375.257,E2 -6375.257} C_VEL
LIN {X 0,Y 489.644,Z 466.366,A -85,B 0,C 180,E1 -6376.512,E2 -6376.512} C_VEL
LIN {X 0,Y 489.137,Z 475.438,A -85,B 0,C 180,E1 -6377.873,E2 -6377.873} C_VEL
LIN {X 0,Y 488.703,Z 484.073,A -85,B 0,C 180,E1 -6379.434,E2 -6379.434} C_VEL
LIN {X 0,Y 488.442,Z 490.705,A -85,B 0,C 180,E1 -6380.893,E2 -6380.893} C_VEL
LIN {X 0,Y 488.203,Z 496.849,A -85,B 0,C 180,E1 -6382.555,E2 -6382.555} C_VEL
LIN {X 0,Y 488.118,Z 501.589,A -85,B 0,C 180,E1 -6384.215,E2 -6384.215} C_VEL
LIN {X 0,Y 488.015,Z 505.067,A -85,B 0,C 180,E1 -6385.87,E2 -6385.87} C_VEL
LIN {X 0,Y 487.985,Z 507.367,A -85,B 0,C 180,E1 -6387.523,E2 -6387.523} C_VEL
LIN {X 0,Y 487.831,Z 508.551,A -85,B 0,C 180,E1 -6389.174,E2 -6389.174} C_VEL
LIN {X 0,Y 487.831,Z 508.569,A -85,B 0,C 180,E1 -6390.825,E2 -6390.825} C_VEL
LIN {X 0,Y 487.985,Z 507.457,A -85,B 0,C 180,E1 -6392.476,E2 -6392.476} C_VEL
LIN {X 0,Y 488.015,Z 505.228,A -85,B 0,C 180,E1 -6394.129,E2 -6394.129} C_VEL
LIN {X 0,Y 488.101,Z 501.818,A -85,B 0,C 180,E1 -6395.784,E2 -6395.784} C_VEL
LIN {X 0,Y 488.202,Z 497.151,A -85,B 0,C 180,E1 -6397.444,E2 -6397.444} C_VEL
LIN {X 0,Y 488.432,Z 491.096,A -85,B 0,C 180,E1 -6399.107,E2 -6399.107} C_VEL
LIN {X 0,Y 488.749,Z 483.469,A -85,B 0,C 180,E1 -6400.774,E2 -6400.774} C_VEL
LIN {X 0,Y 489.153,Z 474.858,A -85,B 0,C 180,E1 -6402.311,E2 -6402.311} C_VEL
LIN {X 0,Y 489.719,Z 465.519,A -85,B 0,C 180,E1 -6403.697,E2 -6403.697} C_VEL
LIN {X 0,Y 490.295,Z 455.453,A -85,B 0,C 180,E1 -6404.952,E2 -6404.952} C_VEL
LIN {X 0,Y 490.867,Z 444.861,A -85,B 0,C 180,E1 -6406.071,E2 -6406.071} C_VEL
LIN {X 0,Y 491.631,Z 432.71,A -85,B 0,C 180,E1 -6407.148,E2 -6407.148} C_VEL
LIN {X 0,Y 492.299,Z 419.921,A -85,B 0,C 180,E1 -6408.089,E2 -6408.089} C_VEL
LIN {X 0,Y 492.923,Z 405.888,A -85,B 0,C 180,E1 -6408.927,E2 -6408.927} C_VEL
LIN {X 0,Y 493.529,Z 390.885,A -85,B 0,C 180,E1 -6409.622,E2 -6409.622} C_VEL
LIN {X 0,Y 493.801,Z 377.37,A -85,B 0,C 180,E1 -6410.099,E2 -6410.099} C_VEL
LIN {X 0,Y 490.715,Z 366.216,A -85,B 0,C 180,E1 -6410.534,E2 -6410.534} C_VEL
LIN {X 0,Y 488.041,Z 357.594,A -85,B 0,C 180,E1 -6410.834,E2 -6410.834} C_VEL
LIN {X 0,Y 488.081,Z 354.531,A -85,B 0,C 180,E1 -6413.777,E2 -6413.777} C_VEL
LIN {X 0,Y 488.177,Z 351.507,A -85,B 0,C 180,E1 -6416.801,E2 -6416.801} C_VEL
LIN {X 0,Y 488.208,Z 349.155,A -85,B 0,C 180,E1 -6419.304,E2 -6419.304} C_VEL
LIN {X 0,Y 488.286,Z 346.513,A -85,B 0,C 180,E1 -6422.177,E2 -6422.177} C_VEL
LIN {X 0,Y 488.367,Z 343.836,A -85,B 0,C 180,E1 -6425.143,E2 -6425.143} C_VEL
LIN {X 0,Y 488.385,Z 341.086,A -85,B 0,C 180,E1 -6428.227,E2 -6428.227} C_VEL
LIN {X 0,Y 488.409,Z 340.276,A -85,B 0,C 180,E1 -6429.282,E2 -6429.282} C_VEL
LIN {X 0,Y 488.629,Z 340.245,A -85,B 0,C 180,E1 -6431.589,E2 -6431.589} C_VEL
LIN {X 0,Y 488.699,Z 340.234,A -85,B 0,C 180,E1 -6434.024,E2 -6434.024} C_VEL
LIN {X 0,Y 488.708,Z 340.234,A -85,B 0,C 180,E1 -6437.173,E2 -6437.173} C_VEL
LIN {X 0,Y 488.731,Z 340.231,A -85,B 0,C 180,E1 -6439.676,E2 -6439.676} C_VEL
LIN {X 0,Y 488.682,Z 340.236,A -85,B 0,C 180,E1 -6442.841,E2 -6442.841} C_VEL
LIN {X 0,Y 488.734,Z 340.227,A -85,B 0,C 180,E1 -6445.887,E2 -6445.887} C_VEL
LIN {X 0,Y 488.695,Z 340.235,A -85,B 0,C 180,E1 -6448.82,E2 -6448.82} C_VEL
LIN {X 0,Y 488.746,Z 340.225,A -85,B 0,C 180,E1 -6451.671,E2 -6451.671} C_VEL
LIN {X 0,Y 488.75,Z 340.229,A -85,B 0,C 180,E1 -6454.444,E2 -6454.444} C_VEL
LIN {X 0,Y 488.719,Z 340.234,A -85,B 0,C 180,E1 -6457.153,E2 -6457.153} C_VEL
LIN {X 0,Y 488.727,Z 340.221,A -85,B 0,C 180,E1 -6459.81,E2 -6459.81} C_VEL
LIN {X 0,Y 488.734,Z 340.231,A -85,B 0,C 180,E1 -6462.423,E2 -6462.423} C_VEL
LIN {X 0,Y 488.76,Z 340.226,A -85,B 0,C 180,E1 -6464.999,E2 -6464.999} C_VEL
LIN {X 0,Y 488.828,Z 340.217,A -85,B 0,C 180,E1 -6468.388,E2 -6468.388} C_VEL
LIN {X 0,Y 488.816,Z 340.219,A -85,B 0,C 180,E1 -6471.734,E2 -6471.734} C_VEL
LIN {X 0,Y 488.855,Z 340.219,A -85,B 0,C 180,E1 -6474.224,E2 -6474.224} C_VEL
LIN {X 0,Y 488.96,Z 340.204,A -85,B 0,C 180,E1 -6477.529,E2 -6477.529} C_VEL
LIN {X 0,Y 488.953,Z 340.204,A -85,B 0,C 180,E1 -6480.823,E2 -6480.823} C_VEL
LIN {X 0,Y 488.96,Z 340.202,A -85,B 0,C 180,E1 -6482.471,E2 -6482.471} C_VEL
LIN {X 0,Y 488.854,Z 340.216,A -85,B 0,C 180,E1 -6485.776,E2 -6485.776} C_VEL
LIN {X 0,Y 488.815,Z 340.221,A -85,B 0,C 180,E1 -6488.266,E2 -6488.266} C_VEL
LIN {X 0,Y 488.806,Z 340.221,A -85,B 0,C 180,E1 -6491.612,E2 -6491.612} C_VEL
LIN {X 0,Y 488.76,Z 340.227,A -85,B 0,C 180,E1 -6495,E2 -6495} C_VEL
LIN {X 0,Y 488.753,Z 340.23,A -85,B 0,C 180,E1 -6498.442,E2 -6498.442} C_VEL
LIN {X 0,Y 488.706,Z 340.234,A -85,B 0,C 180,E1 -6501.071,E2 -6501.071} C_VEL
LIN {X 0,Y 488.691,Z 340.237,A -85,B 0,C 180,E1 -6503.745,E2 -6503.745} C_VEL
LIN {X 0,Y 488.79,Z 340.225,A -85,B 0,C 180,E1 -6506.944,E2 -6506.944} C_VEL
LIN {X 0,Y 488.717,Z 340.235,A -85,B 0,C 180,E1 -6510.365,E2 -6510.365} C_VEL
LIN {X 0,Y 488.734,Z 340.234,A -85,B 0,C 180,E1 -6513.485,E2 -6513.485} C_VEL
LIN {X 0,Y 488.687,Z 340.239,A -85,B 0,C 180,E1 -6516.356,E2 -6516.356} C_VEL
LIN {X 0,Y 488.7,Z 340.236,A -85,B 0,C 180,E1 -6519.254,E2 -6519.254} C_VEL
LIN {X 0,Y 488.707,Z 340.238,A -85,B 0,C 180,E1 -6521.6,E2 -6521.6} C_VEL
LIN {X 0,Y 488.69,Z 340.289,A -85,B 0,C 180,E1 -6523.751,E2 -6523.751} C_VEL
LIN {X 0,Y 489.534,Z 345.239,A -85,B 0,C 180,E1 -6526.441,E2 -6526.441} C_VEL
LIN {X 0,Y 490.066,Z 349.78,A -85,B 0,C 180,E1 -6528.725,E2 -6528.725} C_VEL
LIN {X 0,Y 489.922,Z 354.329,A -85,B 0,C 180,E1 -6530.863,E2 -6530.863} C_VEL
LIN {X 0,Y 489.675,Z 361.269,A -85,B 0,C 180,E1 -6533.954,E2 -6533.954} C_VEL
LIN {X 0,Y 489.34,Z 369.514,A -85,B 0,C 180,E1 -6537.413,E2 -6537.413} C_VEL
LIN {X 0,Y 489.116,Z 377.787,A -85,B 0,C 180,E1 -6540.756,E2 -6540.756} C_VEL
LIN {X 0,Y 488.824,Z 386.051,A -85,B 0,C 180,E1 -6543.992,E2 -6543.992} C_VEL
LIN {X 0,Y 488.562,Z 394.219,A -85,B 0,C 180,E1 -6547.146,E2 -6547.146} C_VEL
LIN {X 0,Y 488.468,Z 399.517,A -85,B 0,C 180,E1 -6549.189,E2 -6549.189} C_VEL
LIN {X 0,Y 492.542,Z 417.595,A -85,B 0,C 180,E1 -6549.74,E2 -6549.74} C_VEL
LIN {X 0,Y 493.702,Z 423.522,A -85,B 0,C 180,E1 -6549.962,E2 -6549.962} C_VEL
LIN {X 0,Y 493.222,Z 437.224,A -85,B 0,C 180,E1 -6550.442,E2 -6550.442} C_VEL
LIN {X 0,Y 492.66,Z 450.759,A -85,B 0,C 180,E1 -6551.063,E2 -6551.063} C_VEL
LIN {X 0,Y 491.923,Z 465.119,A -85,B 0,C 180,E1 -6551.897,E2 -6551.897} C_VEL
LIN {X 0,Y 491.263,Z 478.205,A -85,B 0,C 180,E1 -6552.839,E2 -6552.839} C_VEL
LIN {X 0,Y 490.634,Z 489.672,A -85,B 0,C 180,E1 -6553.826,E2 -6553.826} C_VEL
LIN {X 0,Y 489.94,Z 501.497,A -85,B 0,C 180,E1 -6555.037,E2 -6555.037} C_VEL
LIN {X 0,Y 489.405,Z 511.811,A -85,B 0,C 180,E1 -6556.294,E2 -6556.294} C_VEL
LIN {X 0,Y 488.868,Z 522.115,A -85,B 0,C 180,E1 -6557.792,E2 -6557.792} C_VEL
LIN {X 0,Y 488.536,Z 531.384,A -85,B 0,C 180,E1 -6559.431,E2 -6559.431} C_VEL
LIN {X 0,Y 488.253,Z 538.171,A -85,B 0,C 180,E1 -6560.89,E2 -6560.89} C_VEL
LIN {X 0,Y 488.068,Z 544.446,A -85,B 0,C 180,E1 -6562.554,E2 -6562.554} C_VEL
LIN {X 0,Y 487.999,Z 549.303,A -85,B 0,C 180,E1 -6564.214,E2 -6564.214} C_VEL
LIN {X 0,Y 487.898,Z 552.859,A -85,B 0,C 180,E1 -6565.87,E2 -6565.87} C_VEL
LIN {X 0,Y 487.883,Z 555.2,A -85,B 0,C 180,E1 -6567.524,E2 -6567.524} C_VEL
LIN {X 0,Y 487.831,Z 556.376,A -85,B 0,C 180,E1 -6569.175,E2 -6569.175} C_VEL
LIN {X 0,Y 487.831,Z 556.375,A -85,B 0,C 180,E1 -6570.826,E2 -6570.826} C_VEL
LIN {X 0,Y 487.883,Z 555.195,A -85,B 0,C 180,E1 -6572.477,E2 -6572.477} C_VEL
LIN {X 0,Y 487.898,Z 552.853,A -85,B 0,C 180,E1 -6574.131,E2 -6574.131} C_VEL
LIN {X 0,Y 488.01,Z 549.303,A -85,B 0,C 180,E1 -6575.786,E2 -6575.786} C_VEL
LIN {X 0,Y 488.07,Z 544.447,A -85,B 0,C 180,E1 -6577.447,E2 -6577.447} C_VEL
LIN {X 0,Y 488.253,Z 538.165,A -85,B 0,C 180,E1 -6579.111,E2 -6579.111} C_VEL
LIN {X 0,Y 488.618,Z 530.282,A -85,B 0,C 180,E1 -6580.777,E2 -6580.777} C_VEL
LIN {X 0,Y 488.856,Z 522.074,A -85,B 0,C 180,E1 -6582.215,E2 -6582.215} C_VEL
LIN {X 0,Y 489.41,Z 511.807,A -85,B 0,C 180,E1 -6583.706,E2 -6583.706} C_VEL
LIN {X 0,Y 489.905,Z 501.49,A -85,B 0,C 180,E1 -6584.965,E2 -6584.965} C_VEL
LIN {X 0,Y 490.665,Z 489.548,A -85,B 0,C 180,E1 -6586.187,E2 -6586.187} C_VEL
LIN {X 0,Y 491.298,Z 476.9,A -85,B 0,C 180,E1 -6587.268,E2 -6587.268} C_VEL
LIN {X 0,Y 492.029,Z 463.512,A -85,B 0,C 180,E1 -6588.208,E2 -6588.208} C_VEL
LIN {X 0,Y 492.691,Z 450.744,A -85,B 0,C 180,E1 -6588.937,E2 -6588.937} C_VEL
LIN {X 0,Y 493.211,Z 436.154,A -85,B 0,C 180,E1 -6589.603,E2 -6589.603} C_VEL
LIN {X 0,Y 493.627,Z 422.608,A -85,B 0,C 180,E1 -6590.069,E2 -6590.069} C_VEL
LIN {X 0,Y 490.157,Z 407.046,A -85,B 0,C 180,E1 -6590.599,E2 -6590.599} C_VEL
LIN {X 0,Y 488.462,Z 399.526,A -85,B 0,C 180,E1 -6590.807,E2 -6590.807} C_VEL
LIN {X 0,Y 488.612,Z 391.879,A -85,B 0,C 180,E1 -6593.75,E2 -6593.75} C_VEL
LIN {X 0,Y 488.86,Z 384.854,A -85,B 0,C 180,E1 -6596.466,E2 -6596.466} C_VEL
LIN {X 0,Y 489.117,Z 377.756,A -85,B 0,C 180,E1 -6599.245,E2 -6599.245} C_VEL
LIN {X 0,Y 489.326,Z 369.44,A -85,B 0,C 180,E1 -6602.589,E2 -6602.589} C_VEL
LIN {X 0,Y 489.607,Z 362.408,A -85,B 0,C 180,E1 -6605.546,E2 -6605.546} C_VEL
LIN {X 0,Y 489.847,Z 356.59,A -85,B 0,C 180,E1 -6608.093,E2 -6608.093} C_VEL
LIN {X 0,Y 490.045,Z 351.275,A -85,B 0,C 180,E1 -6610.527,E2 -6610.527} C_VEL
LIN {X 0,Y 489.87,Z 347.438,A -85,B 0,C 180,E1 -6612.4,E2 -6612.4} C_VEL
LIN {X 0,Y 489.024,Z 342.08,A -85,B 0,C 180,E1 -6615.235,E2 -6615.235} C_VEL
LIN {X 0,Y 488.688,Z 340.236,A -85,B 0,C 180,E1 -6616.346,E2 -6616.346} C_VEL
LIN {X 0,Y 488.735,Z 340.232,A -85,B 0,C 180,E1 -6619.677,E2 -6619.677} C_VEL
LIN {X 0,Y 488.685,Z 340.241,A -85,B 0,C 180,E1 -6622.842,E2 -6622.842} C_VEL
LIN {X 0,Y 488.737,Z 340.234,A -85,B 0,C 180,E1 -6625.888,E2 -6625.888} C_VEL
LIN {X 0,Y 488.694,Z 340.237,A -85,B 0,C 180,E1 -6628.821,E2 -6628.821} C_VEL
LIN {X 0,Y 488.748,Z 340.229,A -85,B 0,C 180,E1 -6631.672,E2 -6631.672} C_VEL
LIN {X 0,Y 488.743,Z 340.23,A -85,B 0,C 180,E1 -6634.444,E2 -6634.444} C_VEL
LIN {X 0,Y 488.725,Z 340.235,A -85,B 0,C 180,E1 -6637.153,E2 -6637.153} C_VEL
LIN {X 0,Y 488.728,Z 340.234,A -85,B 0,C 180,E1 -6639.811,E2 -6639.811} C_VEL
LIN {X 0,Y 488.737,Z 340.231,A -85,B 0,C 180,E1 -6642.424,E2 -6642.424} C_VEL
LIN {X 0,Y 488.766,Z 340.229,A -85,B 0,C 180,E1 -6645,E2 -6645} C_VEL
LIN {X 0,Y 488.809,Z 340.222,A -85,B 0,C 180,E1 -6648.388,E2 -6648.388} C_VEL
LIN {X 0,Y 488.821,Z 340.221,A -85,B 0,C 180,E1 -6651.734,E2 -6651.734} C_VEL
LIN {X 0,Y 488.858,Z 340.216,A -85,B 0,C 180,E1 -6654.224,E2 -6654.224} C_VEL
LIN {X 0,Y 488.965,Z 340.201,A -85,B 0,C 180,E1 -6657.529,E2 -6657.529} C_VEL
LIN {X 0,Y 488.958,Z 340.202,A -85,B 0,C 180,E1 -6660.824,E2 -6660.824} C_VEL
LIN {X 0,Y 488.964,Z 340.203,A -85,B 0,C 180,E1 -6662.471,E2 -6662.471} C_VEL
LIN {X 0,Y 488.86,Z 340.218,A -85,B 0,C 180,E1 -6665.776,E2 -6665.776} C_VEL
LIN {X 0,Y 488.822,Z 340.219,A -85,B 0,C 180,E1 -6668.266,E2 -6668.266} C_VEL
LIN {X 0,Y 488.809,Z 340.217,A -85,B 0,C 180,E1 -6671.612,E2 -6671.612} C_VEL
LIN {X 0,Y 488.766,Z 340.226,A -85,B 0,C 180,E1 -6675,E2 -6675} C_VEL
LIN {X 0,Y 488.759,Z 340.225,A -85,B 0,C 180,E1 -6678.442,E2 -6678.442} C_VEL
LIN {X 0,Y 488.71,Z 340.226,A -85,B 0,C 180,E1 -6681.071,E2 -6681.071} C_VEL
LIN {X 0,Y 488.683,Z 340.237,A -85,B 0,C 180,E1 -6683.746,E2 -6683.746} C_VEL
LIN {X 0,Y 488.795,Z 340.219,A -85,B 0,C 180,E1 -6686.944,E2 -6686.944} C_VEL
LIN {X 0,Y 488.713,Z 340.237,A -85,B 0,C 180,E1 -6690.363,E2 -6690.363} C_VEL
LIN {X 0,Y 488.739,Z 340.226,A -85,B 0,C 180,E1 -6693.484,E2 -6693.484} C_VEL
LIN {X 0,Y 488.692,Z 340.24,A -85,B 0,C 180,E1 -6696.355,E2 -6696.355} C_VEL
LIN {X 0,Y 488.705,Z 340.237,A -85,B 0,C 180,E1 -6699.254,E2 -6699.254} C_VEL
LIN {X 0,Y 488.71,Z 340.234,A -85,B 0,C 180,E1 -6701.6,E2 -6701.6} C_VEL
LIN {X 0,Y 488.715,Z 340.234,A -85,B 0,C 180,E1 -6704.801,E2 -6704.801} C_VEL
LIN {X 0,Y 488.674,Z 340.241,A -85,B 0,C 180,E1 -6707.472,E2 -6707.472} C_VEL
LIN {X 0,Y 488.541,Z 340.259,A -85,B 0,C 180,E1 -6709.68,E2 -6709.68} C_VEL
LIN {X 0,Y 488.405,Z 340.321,A -85,B 0,C 180,E1 -6710.991,E2 -6710.991} C_VEL
LIN {X 0,Y 488.368,Z 342.833,A -85,B 0,C 180,E1 -6713.841,E2 -6713.841} C_VEL
LIN {X 0,Y 488.329,Z 345.51,A -85,B 0,C 180,E1 -6716.845,E2 -6716.845} C_VEL
LIN {X 0,Y 488.259,Z 348.181,A -85,B 0,C 180,E1 -6719.749,E2 -6719.749} C_VEL
LIN {X 0,Y 488.168,Z 350.799,A -85,B 0,C 180,E1 -6722.568,E2 -6722.568} C_VEL
LIN {X 0,Y 488.148,Z 352.433,A -85,B 0,C 180,E1 -6724.226,E2 -6724.226} C_VEL
LIN {X 0,Y 487.484,Z 353.178,A -85,B 0,C 180,E1 -6724.908,E2 -6724.908} C_VEL
LIN {X 0,Y 484.603,Z 354.56,A -85,B 0,C 180,E1 -6726.013,E2 -6726.013} C_VEL
LIN {X 0,Y 482.147,Z 355.698,A -85,B 0,C 180,E1 -6726.904,E2 -6726.904} C_VEL
LIN {X 0,Y 481.074,Z 356.516,A -85,B 0,C 180,E1 -6727.593,E2 -6727.593} C_VEL
LIN {X 0,Y 480.977,Z 356.773,A -85,B 0,C 180,E1 -6727.826,E2 -6727.826} C_VEL
LIN {X 0,Y 480.972,Z 358.001,A -85,B 0,C 180,E1 -6728.95,E2 -6728.95} C_VEL
LIN {X 0,Y 485.812,Z 373.441,A -85,B 0,C 180,E1 -6729.514,E2 -6729.514} C_VEL
LIN {X 0,Y 487.207,Z 378.96,A -85,B 0,C 180,E1 -6729.744,E2 -6729.744} C_VEL
LIN {X 0,Y 486.815,Z 393.923,A -85,B 0,C 180,E1 -6730.301,E2 -6730.301} C_VEL
LIN {X 0,Y 486.124,Z 408.531,A -85,B 0,C 180,E1 -6731.017,E2 -6731.017} C_VEL
LIN {X 0,Y 485.475,Z 422.09,A -85,B 0,C 180,E1 -6731.865,E2 -6731.865} C_VEL
LIN {X 0,Y 484.717,Z 434.553,A -85,B 0,C 180,E1 -6732.817,E2 -6732.817} C_VEL
LIN {X 0,Y 483.908,Z 447.163,A -85,B 0,C 180,E1 -6733.981,E2 -6733.981} C_VEL
LIN {X 0,Y 483.211,Z 458.584,A -85,B 0,C 180,E1 -6735.254,E2 -6735.254} C_VEL
LIN {X 0,Y 482.634,Z 468.188,A -85,B 0,C 180,E1 -6736.527,E2 -6736.527} C_VEL
LIN {X 0,Y 482.097,Z 477.488,A -85,B 0,C 180,E1 -6737.991,E2 -6737.991} C_VEL
LIN {X 0,Y 481.641,Z 485.422,A -85,B 0,C 180,E1 -6739.49,E2 -6739.49} C_VEL
LIN {X 0,Y 481.334,Z 492.722,A -85,B 0,C 180,E1 -6741.181,E2 -6741.181} C_VEL
LIN {X 0,Y 481.108,Z 498.515,A -85,B 0,C 180,E1 -6742.867,E2 -6742.867} C_VEL
LIN {X 0,Y 481.055,Z 501.939,A -85,B 0,C 180,E1 -6744.13,E2 -6744.13} C_VEL
LIN {X 0,Y 480.936,Z 505.416,A -85,B 0,C 180,E1 -6745.81,E2 -6745.81} C_VEL
LIN {X 0,Y 480.905,Z 507.715,A -85,B 0,C 180,E1 -6747.487,E2 -6747.487} C_VEL
LIN {X 0,Y 480.757,Z 508.898,A -85,B 0,C 180,E1 -6749.162,E2 -6749.162} C_VEL
LIN {X 0,Y 480.757,Z 508.916,A -85,B 0,C 180,E1 -6750.837,E2 -6750.837} C_VEL
LIN {X 0,Y 480.906,Z 507.804,A -85,B 0,C 180,E1 -6752.512,E2 -6752.512} C_VEL
LIN {X 0,Y 480.935,Z 505.575,A -85,B 0,C 180,E1 -6754.19,E2 -6754.19} C_VEL
LIN {X 0,Y 481.04,Z 502.165,A -85,B 0,C 180,E1 -6755.87,E2 -6755.87} C_VEL
LIN {X 0,Y 481.147,Z 497.497,A -85,B 0,C 180,E1 -6757.554,E2 -6757.554} C_VEL
LIN {X 0,Y 481.414,Z 491.442,A -85,B 0,C 180,E1 -6759.24,E2 -6759.24} C_VEL
LIN {X 0,Y 481.764,Z 483.814,A -85,B 0,C 180,E1 -6760.932,E2 -6760.932} C_VEL
LIN {X 0,Y 482.16,Z 475.65,A -85,B 0,C 180,E1 -6762.42,E2 -6762.42} C_VEL
LIN {X 0,Y 482.811,Z 465.863,A -85,B 0,C 180,E1 -6763.897,E2 -6763.897} C_VEL
LIN {X 0,Y 483.429,Z 455.796,A -85,B 0,C 180,E1 -6765.169,E2 -6765.169} C_VEL
LIN {X 0,Y 484.099,Z 444.312,A -85,B 0,C 180,E1 -6766.393,E2 -6766.393} C_VEL
LIN {X 0,Y 484.891,Z 431.771,A -85,B 0,C 180,E1 -6767.502,E2 -6767.502} C_VEL
LIN {X 0,Y 485.661,Z 418.687,A -85,B 0,C 180,E1 -6768.454,E2 -6768.454} C_VEL
LIN {X 0,Y 486.231,Z 406.223,A -85,B 0,C 180,E1 -6769.197,E2 -6769.197} C_VEL
LIN {X 0,Y 486.841,Z 391.856,A -85,B 0,C 180,E1 -6769.876,E2 -6769.876} C_VEL
LIN {X 0,Y 487.203,Z 379.097,A -85,B 0,C 180,E1 -6770.341,E2 -6770.341} C_VEL
LIN {X 0,Y 483.831,Z 366.962,A -85,B 0,C 180,E1 -6770.83,E2 -6770.83} C_VEL
LIN {X 0,Y 480.97,Z 357.996,A -85,B 0,C 180,E1 -6771.141,E2 -6771.141} C_VEL
LIN {X 0,Y 481.015,Z 354.835,A -85,B 0,C 180,E1 -6774.148,E2 -6774.148} C_VEL
LIN {X 0,Y 481.124,Z 352.015,A -85,B 0,C 180,E1 -6776.994,E2 -6776.994} C_VEL
LIN {X 0,Y 481.15,Z 349.422,A -85,B 0,C 180,E1 -6779.777,E2 -6779.777} C_VEL
LIN {X 0,Y 481.252,Z 346.76,A -85,B 0,C 180,E1 -6782.706,E2 -6782.706} C_VEL
LIN {X 0,Y 481.309,Z 344.061,A -85,B 0,C 180,E1 -6785.737,E2 -6785.737} C_VEL
LIN {X 0,Y 481.335,Z 342.09,A -85,B 0,C 180,E1 -6787.958,E2 -6787.958} C_VEL
LIN {X 0,Y 481.374,Z 341.152,A -85,B 0,C 180,E1 -6789.304,E2 -6789.304} C_VEL
LIN {X 0,Y 481.615,Z 341.115,A -85,B 0,C 180,E1 -6792.164,E2 -6792.164} C_VEL
LIN {X 0,Y 481.659,Z 341.114,A -85,B 0,C 180,E1 -6794.457,E2 -6794.457} C_VEL
LIN {X 0,Y 481.647,Z 341.116,A -85,B 0,C 180,E1 -6797.839,E2 -6797.839} C_VEL
LIN {X 0,Y 481.68,Z 341.113,A -85,B 0,C 180,E1 -6800.651,E2 -6800.651} C_VEL
LIN {X 0,Y 481.631,Z 341.116,A -85,B 0,C 180,E1 -6803.375,E2 -6803.375} C_VEL
LIN {X 0,Y 481.708,Z 341.103,A -85,B 0,C 180,E1 -6806.33,E2 -6806.33} C_VEL
LIN {X 0,Y 481.657,Z 341.113,A -85,B 0,C 180,E1 -6809.415,E2 -6809.415} C_VEL
LIN {X 0,Y 481.702,Z 341.101,A -85,B 0,C 180,E1 -6812.168,E2 -6812.168} C_VEL
LIN {X 0,Y 481.717,Z 341.103,A -85,B 0,C 180,E1 -6814.97,E2 -6814.97} C_VEL
LIN {X 0,Y 481.649,Z 341.11,A -85,B 0,C 180,E1 -6817.705,E2 -6817.705} C_VEL
LIN {X 0,Y 481.706,Z 341.1,A -85,B 0,C 180,E1 -6820.393,E2 -6820.393} C_VEL
LIN {X 0,Y 481.691,Z 341.108,A -85,B 0,C 180,E1 -6823.034,E2 -6823.034} C_VEL
LIN {X 0,Y 481.688,Z 341.102,A -85,B 0,C 180,E1 -6825.639,E2 -6825.639} C_VEL
LIN {X 0,Y 481.793,Z 341.093,A -85,B 0,C 180,E1 -6828.216,E2 -6828.216} C_VEL
LIN {X 0,Y 481.762,Z 341.098,A -85,B 0,C 180,E1 -6831.612,E2 -6831.612} C_VEL
LIN {X 0,Y 481.816,Z 341.096,A -85,B 0,C 180,E1 -6834.139,E2 -6834.139} C_VEL
LIN {X 0,Y 481.927,Z 341.08,A -85,B 0,C 180,E1 -6837.492,E2 -6837.492} C_VEL
LIN {X 0,Y 481.904,Z 341.082,A -85,B 0,C 180,E1 -6840.836,E2 -6840.836} C_VEL
LIN {X 0,Y 481.927,Z 341.078,A -85,B 0,C 180,E1 -6842.507,E2 -6842.507} C_VEL
LIN {X 0,Y 481.815,Z 341.094,A -85,B 0,C 180,E1 -6845.86,E2 -6845.86} C_VEL
LIN {X 0,Y 481.761,Z 341.099,A -85,B 0,C 180,E1 -6848.388,E2 -6848.388} C_VEL
LIN {X 0,Y 481.751,Z 341.1,A -85,B 0,C 180,E1 -6851.785,E2 -6851.785} C_VEL
LIN {X 0,Y 481.741,Z 341.103,A -85,B 0,C 180,E1 -6855.224,E2 -6855.224} C_VEL
LIN {X 0,Y 481.71,Z 341.108,A -85,B 0,C 180,E1 -6858.722,E2 -6858.722} C_VEL
LIN {X 0,Y 481.646,Z 341.116,A -85,B 0,C 180,E1 -6861.395,E2 -6861.395} C_VEL
LIN {X 0,Y 481.675,Z 341.112,A -85,B 0,C 180,E1 -6864.113,E2 -6864.113} C_VEL
LIN {X 0,Y 481.745,Z 341.103,A -85,B 0,C 180,E1 -6867.139,E2 -6867.139} C_VEL
LIN {X 0,Y 481.686,Z 341.11,A -85,B 0,C 180,E1 -6869.741,E2 -6869.741} C_VEL
LIN {X 0,Y 481.671,Z 341.112,A -85,B 0,C 180,E1 -6872.674,E2 -6872.674} C_VEL
LIN {X 0,Y 481.641,Z 341.116,A -85,B 0,C 180,E1 -6875.709,E2 -6875.709} C_VEL
LIN {X 0,Y 481.67,Z 341.111,A -85,B 0,C 180,E1 -6878.859,E2 -6878.859} C_VEL
LIN {X 0,Y 481.651,Z 341.115,A -85,B 0,C 180,E1 -6881.913,E2 -6881.913} C_VEL
LIN {X 0,Y 481.669,Z 341.225,A -85,B 0,C 180,E1 -6883.44,E2 -6883.44} C_VEL
LIN {X 0,Y 482.505,Z 346.089,A -85,B 0,C 180,E1 -6886.136,E2 -6886.136} C_VEL
LIN {X 0,Y 483.078,Z 350.766,A -85,B 0,C 180,E1 -6888.552,E2 -6888.552} C_VEL
LIN {X 0,Y 483.014,Z 354.731,A -85,B 0,C 180,E1 -6890.459,E2 -6890.459} C_VEL
LIN {X 0,Y 482.672,Z 362.254,A -85,B 0,C 180,E1 -6893.864,E2 -6893.864} C_VEL
LIN {X 0,Y 482.322,Z 370.475,A -85,B 0,C 180,E1 -6897.376,E2 -6897.376} C_VEL
LIN {X 0,Y 482.044,Z 377.541,A -85,B 0,C 180,E1 -6900.284,E2 -6900.284} C_VEL
LIN {X 0,Y 481.838,Z 384.603,A -85,B 0,C 180,E1 -6903.118,E2 -6903.118} C_VEL
LIN {X 0,Y 481.575,Z 392.77,A -85,B 0,C 180,E1 -6906.339,E2 -6906.339} C_VEL
LIN {X 0,Y 481.411,Z 399.211,A -85,B 0,C 180,E1 -6908.875,E2 -6908.875} C_VEL
LIN {X 0,Y 485.273,Z 416.252,A -85,B 0,C 180,E1 -6909.398,E2 -6909.398} C_VEL
LIN {X 0,Y 486.995,Z 424.507,A -85,B 0,C 180,E1 -6909.714,E2 -6909.714} C_VEL
LIN {X 0,Y 486.462,Z 438.594,A -85,B 0,C 180,E1 -6910.232,E2 -6910.232} C_VEL
LIN {X 0,Y 485.797,Z 452.405,A -85,B 0,C 180,E1 -6910.895,E2 -6910.895} C_VEL
LIN {X 0,Y 485.028,Z 466.358,A -85,B 0,C 180,E1 -6911.74,E2 -6911.74} C_VEL
LIN {X 0,Y 484.323,Z 479.153,A -85,B 0,C 180,E1 -6912.694,E2 -6912.694} C_VEL
LIN {X 0,Y 483.617,Z 491.713,A -85,B 0,C 180,E1 -6913.825,E2 -6913.825} C_VEL
LIN {X 0,Y 482.889,Z 502.944,A -85,B 0,C 180,E1 -6915.029,E2 -6915.029} C_VEL
LIN {X 0,Y 482.342,Z 512.989,A -85,B 0,C 180,E1 -6916.304,E2 -6916.304} C_VEL
LIN {X 0,Y 481.758,Z 522.876,A -85,B 0,C 180,E1 -6917.798,E2 -6917.798} C_VEL
LIN {X 0,Y 481.504,Z 531.033,A -85,B 0,C 180,E1 -6919.275,E2 -6919.275} C_VEL
LIN {X 0,Y 481.175,Z 537.82,A -85,B 0,C 180,E1 -6920.755,E2 -6920.755} C_VEL
LIN {X 0,Y 480.993,Z 544.096,A -85,B 0,C 180,E1 -6922.444,E2 -6922.444} C_VEL
LIN {X 0,Y 480.903,Z 548.953,A -85,B 0,C 180,E1 -6924.129,E2 -6924.129} C_VEL
LIN {X 0,Y 480.801,Z 552.51,A -85,B 0,C 180,E1 -6925.809,E2 -6925.809} C_VEL
LIN {X 0,Y 480.799,Z 554.853,A -85,B 0,C 180,E1 -6927.487,E2 -6927.487} C_VEL
LIN {X 0,Y 480.757,Z 556.03,A -85,B 0,C 180,E1 -6929.163,E2 -6929.163} C_VEL
LIN {X 0,Y 480.757,Z 556.029,A -85,B 0,C 180,E1 -6930.838,E2 -6930.838} C_VEL
LIN {X 0,Y 480.799,Z 554.848,A -85,B 0,C 180,E1 -6932.514,E2 -6932.514} C_VEL
LIN {X 0,Y 480.801,Z 552.504,A -85,B 0,C 180,E1 -6934.192,E2 -6934.192} C_VEL
LIN {X 0,Y 480.919,Z 548.953,A -85,B 0,C 180,E1 -6935.872,E2 -6935.872} C_VEL
LIN {X 0,Y 480.994,Z 544.098,A -85,B 0,C 180,E1 -6937.557,E2 -6937.557} C_VEL
LIN {X 0,Y 481.176,Z 537.813,A -85,B 0,C 180,E1 -6939.246,E2 -6939.246} C_VEL
LIN {X 0,Y 481.586,Z 529.932,A -85,B 0,C 180,E1 -6940.936,E2 -6940.936} C_VEL
LIN {X 0,Y 481.818,Z 522.054,A -85,B 0,C 180,E1 -6942.341,E2 -6942.341} C_VEL
LIN {X 0,Y 482.407,Z 511.453,A -85,B 0,C 180,E1 -6943.909,E2 -6943.909} C_VEL
LIN {X 0,Y 482.962,Z 501.138,A -85,B 0,C 180,E1 -6945.185,E2 -6945.185} C_VEL
LIN {X 0,Y 483.713,Z 490.001,A -85,B 0,C 180,E1 -6946.345,E2 -6946.345} C_VEL
LIN {X 0,Y 484.367,Z 477.849,A -85,B 0,C 180,E1 -6947.414,E2 -6947.414} C_VEL
LIN {X 0,Y 485.139,Z 464.753,A -85,B 0,C 180,E1 -6948.366,E2 -6948.366} C_VEL
LIN {X 0,Y 485.816,Z 452.387,A -85,B 0,C 180,E1 -6949.105,E2 -6949.105} C_VEL
LIN {X 0,Y 486.426,Z 438.647,A -85,B 0,C 180,E1 -6949.768,E2 -6949.768} C_VEL
LIN {X 0,Y 486.877,Z 423.405,A -85,B 0,C 180,E1 -6950.325,E2 -6950.325} C_VEL
LIN {X 0,Y 483.61,Z 408.693,A -85,B 0,C 180,E1 -6950.854,E2 -6950.854} C_VEL
LIN {X 0,Y 481.412,Z 399.21,A -85,B 0,C 180,E1 -6951.125,E2 -6951.125} C_VEL
LIN {X 0,Y 481.579,Z 391.589,A -85,B 0,C 180,E1 -6954.119,E2 -6954.119} C_VEL
LIN {X 0,Y 481.845,Z 384.58,A -85,B 0,C 180,E1 -6956.882,E2 -6956.882} C_VEL
LIN {X 0,Y 482.064,Z 377.499,A -85,B 0,C 180,E1 -6959.715,E2 -6959.715} C_VEL
LIN {X 0,Y 482.311,Z 370.388,A -85,B 0,C 180,E1 -6962.626,E2 -6962.626} C_VEL
LIN {X 0,Y 482.615,Z 363.371,A -85,B 0,C 180,E1 -6965.626,E2 -6965.626} C_VEL
LIN {X 0,Y 482.899,Z 356.42,A -85,B 0,C 180,E1 -6968.742,E2 -6968.742} C_VEL
LIN {X 0,Y 483.063,Z 350.693,A -85,B 0,C 180,E1 -6971.451,E2 -6971.451} C_VEL
LIN {X 0,Y 482.503,Z 346.031,A -85,B 0,C 180,E1 -6973.863,E2 -6973.863} C_VEL
LIN {X 0,Y 481.64,Z 341.117,A -85,B 0,C 180,E1 -6976.7,E2 -6976.7} C_VEL
LIN {X 0,Y 481.679,Z 341.114,A -85,B 0,C 180,E1 -6980.06,E2 -6980.06} C_VEL
LIN {X 0,Y 481.632,Z 341.121,A -85,B 0,C 180,E1 -6983.254,E2 -6983.254} C_VEL
LIN {X 0,Y 481.712,Z 341.11,A -85,B 0,C 180,E1 -6986.33,E2 -6986.33} C_VEL
LIN {X 0,Y 481.653,Z 341.115,A -85,B 0,C 180,E1 -6989.418,E2 -6989.418} C_VEL
LIN {X 0,Y 481.703,Z 341.109,A -85,B 0,C 180,E1 -6992.168,E2 -6992.168} C_VEL
LIN {X 0,Y 481.715,Z 341.106,A -85,B 0,C 180,E1 -6994.97,E2 -6994.97} C_VEL
LIN {X 0,Y 481.652,Z 341.113,A -85,B 0,C 180,E1 -6997.705,E2 -6997.705} C_VEL
LIN {X 0,Y 481.709,Z 341.107,A -85,B 0,C 180,E1 -7000.393,E2 -7000.393} C_VEL
LIN {X 0,Y 481.694,Z 341.112,A -85,B 0,C 180,E1 -7003.034,E2 -7003.034} C_VEL
LIN {X 0,Y 481.693,Z 341.11,A -85,B 0,C 180,E1 -7005.639,E2 -7005.639} C_VEL
LIN {X 0,Y 481.754,Z 341.102,A -85,B 0,C 180,E1 -7008.215,E2 -7008.215} C_VEL
LIN {X 0,Y 481.766,Z 341.099,A -85,B 0,C 180,E1 -7011.612,E2 -7011.612} C_VEL
LIN {X 0,Y 481.819,Z 341.093,A -85,B 0,C 180,E1 -7014.14,E2 -7014.14} C_VEL
LIN {X 0,Y 481.931,Z 341.077,A -85,B 0,C 180,E1 -7017.493,E2 -7017.493} C_VEL
LIN {X 0,Y 481.91,Z 341.08,A -85,B 0,C 180,E1 -7020.836,E2 -7020.836} C_VEL
LIN {X 0,Y 481.931,Z 341.079,A -85,B 0,C 180,E1 -7022.508,E2 -7022.508} C_VEL
LIN {X 0,Y 481.821,Z 341.095,A -85,B 0,C 180,E1 -7025.86,E2 -7025.86} C_VEL
LIN {X 0,Y 481.767,Z 341.098,A -85,B 0,C 180,E1 -7028.388,E2 -7028.388} C_VEL
LIN {X 0,Y 481.754,Z 341.095,A -85,B 0,C 180,E1 -7031.785,E2 -7031.785} C_VEL
LIN {X 0,Y 481.746,Z 341.103,A -85,B 0,C 180,E1 -7035.224,E2 -7035.224} C_VEL
LIN {X 0,Y 481.716,Z 341.1,A -85,B 0,C 180,E1 -7038.722,E2 -7038.722} C_VEL
LIN {X 0,Y 481.649,Z 341.11,A -85,B 0,C 180,E1 -7041.395,E2 -7041.395} C_VEL
LIN {X 0,Y 481.664,Z 341.114,A -85,B 0,C 180,E1 -7044.114,E2 -7044.114} C_VEL
LIN {X 0,Y 481.75,Z 341.095,A -85,B 0,C 180,E1 -7047.139,E2 -7047.139} C_VEL
LIN {X 0,Y 481.682,Z 341.108,A -85,B 0,C 180,E1 -7049.741,E2 -7049.741} C_VEL
LIN {X 0,Y 481.675,Z 341.105,A -85,B 0,C 180,E1 -7052.674,E2 -7052.674} C_VEL
LIN {X 0,Y 481.645,Z 341.113,A -85,B 0,C 180,E1 -7055.709,E2 -7055.709} C_VEL
LIN {X 0,Y 481.675,Z 341.11,A -85,B 0,C 180,E1 -7058.859,E2 -7058.859} C_VEL
LIN {X 0,Y 481.656,Z 341.113,A -85,B 0,C 180,E1 -7061.913,E2 -7061.913} C_VEL
LIN {X 0,Y 481.663,Z 341.114,A -85,B 0,C 180,E1 -7064.457,E2 -7064.457} C_VEL
LIN {X 0,Y 481.641,Z 341.119,A -85,B 0,C 180,E1 -7066.852,E2 -7066.852} C_VEL
LIN {X 0,Y 481.5,Z 341.137,A -85,B 0,C 180,E1 -7069.376,E2 -7069.376} C_VEL
LIN {X 0,Y 481.338,Z 341.2,A -85,B 0,C 180,E1 -7071.109,E2 -7071.109} C_VEL
LIN {X 0,Y 481.324,Z 343.222,A -85,B 0,C 180,E1 -7073.425,E2 -7073.425} C_VEL
LIN {X 0,Y 481.275,Z 345.792,A -85,B 0,C 180,E1 -7076.342,E2 -7076.342} C_VEL
LIN {X 0,Y 481.177,Z 348.441,A -85,B 0,C 180,E1 -7079.256,E2 -7079.256} C_VEL
LIN {X 0,Y 481.112,Z 351.076,A -85,B 0,C 180,E1 -7082.131,E2 -7082.131} C_VEL
LIN {X 0,Y 481.084,Z 353.823,A -85,B 0,C 180,E1 -7084.934,E2 -7084.934} C_VEL
LIN {X 0,Y 480.977,Z 356.773,A -85,B 0,C 180,E1 -7087.826,E2 -7087.826} C_VEL
LIN {X 0,Y 480.932,Z 357.849,A -85,B 0,C 180,E1 -7088.19,E2 -7088.19} C_VEL
LIN {X 0,Y 480.839,Z 360.556,A -85,B 0,C 180,E1 -7088.576,E2 -7088.576} C_VEL
LIN {X 0,Y 480.738,Z 363.754,A -85,B 0,C 180,E1 -7088.848,E2 -7088.848} C_VEL
LIN {X 0,Y 480.637,Z 367.31,A -85,B 0,C 180,E1 -7089.048,E2 -7089.048} C_VEL
LIN {X 0,Y 480.729,Z 375.784,A -85,B 0,C 180,E1 -7089.351,E2 -7089.351} C_VEL
LIN {X 0,Y 480.49,Z 384.336,A -85,B 0,C 180,E1 -7089.626,E2 -7089.626} C_VEL
LIN {X 0,Y 479.923,Z 398.776,A -85,B 0,C 180,E1 -7090.22,E2 -7090.22} C_VEL
LIN {X 0,Y 479.273,Z 412.533,A -85,B 0,C 180,E1 -7090.957,E2 -7090.957} C_VEL
LIN {X 0,Y 478.54,Z 425.435,A -85,B 0,C 180,E1 -7091.815,E2 -7091.815} C_VEL
LIN {X 0,Y 477.81,Z 437.441,A -85,B 0,C 180,E1 -7092.781,E2 -7092.781} C_VEL
LIN {X 0,Y 476.953,Z 449.619,A -85,B 0,C 180,E1 -7093.961,E2 -7093.961} C_VEL
LIN {X 0,Y 476.218,Z 460.699,A -85,B 0,C 180,E1 -7095.251,E2 -7095.251} C_VEL
LIN {X 0,Y 475.524,Z 471.457,A -85,B 0,C 180,E1 -7096.757,E2 -7096.757} C_VEL
LIN {X 0,Y 475.029,Z 480.372,A -85,B 0,C 180,E1 -7098.262,E2 -7098.262} C_VEL
LIN {X 0,Y 474.55,Z 487.762,A -85,B 0,C 180,E1 -7099.763,E2 -7099.763} C_VEL
LIN {X 0,Y 474.224,Z 494.664,A -85,B 0,C 180,E1 -7101.477,E2 -7101.477} C_VEL
LIN {X 0,Y 474.005,Z 500.087,A -85,B 0,C 180,E1 -7103.187,E2 -7103.187} C_VEL
LIN {X 0,Y 473.815,Z 504.183,A -85,B 0,C 180,E1 -7104.894,E2 -7104.894} C_VEL
LIN {X 0,Y 473.822,Z 507.057,A -85,B 0,C 180,E1 -7106.598,E2 -7106.598} C_VEL
LIN {X 0,Y 473.757,Z 508.792,A -85,B 0,C 180,E1 -7108.299,E2 -7108.299} C_VEL
LIN {X 0,Y 473.667,Z 509.403,A -85,B 0,C 180,E1 -7110,E2 -7110} C_VEL
LIN {X 0,Y 473.758,Z 508.844,A -85,B 0,C 180,E1 -7111.7,E2 -7111.7} C_VEL
LIN {X 0,Y 473.823,Z 507.18,A -85,B 0,C 180,E1 -7113.401,E2 -7113.401} C_VEL
LIN {X 0,Y 473.811,Z 504.373,A -85,B 0,C 180,E1 -7115.106,E2 -7115.106} C_VEL
LIN {X 0,Y 474.003,Z 500.342,A -85,B 0,C 180,E1 -7116.812,E2 -7116.812} C_VEL
LIN {X 0,Y 474.222,Z 494.999,A -85,B 0,C 180,E1 -7118.522,E2 -7118.522} C_VEL
LIN {X 0,Y 474.515,Z 488.188,A -85,B 0,C 180,E1 -7120.237,E2 -7120.237} C_VEL
LIN {X 0,Y 474.967,Z 480.853,A -85,B 0,C 180,E1 -7121.739,E2 -7121.739} C_VEL
LIN {X 0,Y 475.49,Z 472.015,A -85,B 0,C 180,E1 -7123.244,E2 -7123.244} C_VEL
LIN {X 0,Y 476.088,Z 462.997,A -85,B 0,C 180,E1 -7124.534,E2 -7124.534} C_VEL
LIN {X 0,Y 476.769,Z 452.353,A -85,B 0,C 180,E1 -7125.825,E2 -7125.825} C_VEL
LIN {X 0,Y 477.533,Z 441.469,A -85,B 0,C 180,E1 -7126.937,E2 -7126.937} C_VEL
LIN {X 0,Y 478.256,Z 429.432,A -85,B 0,C 180,E1 -7127.974,E2 -7127.974} C_VEL
LIN {X 0,Y 479.084,Z 415.738,A -85,B 0,C 180,E1 -7128.939,E2 -7128.939} C_VEL
LIN {X 0,Y 479.776,Z 402.558,A -85,B 0,C 180,E1 -7129.689,E2 -7129.689} C_VEL
LIN {X 0,Y 480.369,Z 387.151,A -85,B 0,C 180,E1 -7130.366,E2 -7130.366} C_VEL
LIN {X 0,Y 480.448,Z 380.024,A -85,B 0,C 180,E1 -7130.622,E2 -7130.622} C_VEL
LIN {X 0,Y 476.751,Z 367.294,A -85,B 0,C 180,E1 -7131.154,E2 -7131.154} C_VEL
LIN {X 0,Y 473.912,Z 358.262,A -85,B 0,C 180,E1 -7131.477,E2 -7131.477} C_VEL
LIN {X 0,Y 473.961,Z 355.144,A -85,B 0,C 180,E1 -7134.531,E2 -7134.531} C_VEL
LIN {X 0,Y 474.041,Z 352.372,A -85,B 0,C 180,E1 -7137.361,E2 -7137.361} C_VEL
LIN {X 0,Y 474.103,Z 349.691,A -85,B 0,C 180,E1 -7140.265,E2 -7140.265} C_VEL
LIN {X 0,Y 474.198,Z 347.012,A -85,B 0,C 180,E1 -7143.255,E2 -7143.255} C_VEL
LIN {X 0,Y 474.251,Z 344.29,A -85,B 0,C 180,E1 -7146.353,E2 -7146.353} C_VEL
LIN {X 0,Y 474.27,Z 342.413,A -85,B 0,C 180,E1 -7148.49,E2 -7148.49} C_VEL
LIN {X 0,Y 474.351,Z 342.026,A -85,B 0,C 180,E1 -7149.607,E2 -7149.607} C_VEL
LIN {X 0,Y 474.576,Z 341.992,A -85,B 0,C 180,E1 -7152.23,E2 -7152.23} C_VEL
LIN {X 0,Y 474.62,Z 341.988,A -85,B 0,C 180,E1 -7155.297,E2 -7155.297} C_VEL
LIN {X 0,Y 474.62,Z 341.989,A -85,B 0,C 180,E1 -7158.214,E2 -7158.214} C_VEL
LIN {X 0,Y 474.644,Z 341.988,A -85,B 0,C 180,E1 -7160.454,E2 -7160.454} C_VEL
LIN {X 0,Y 474.593,Z 341.995,A -85,B 0,C 180,E1 -7163.677,E2 -7163.677} C_VEL
LIN {X 0,Y 474.641,Z 341.982,A -85,B 0,C 180,E1 -7166.78,E2 -7166.78} C_VEL
LIN {X 0,Y 474.613,Z 341.994,A -85,B 0,C 180,E1 -7169.77,E2 -7169.77} C_VEL
LIN {X 0,Y 474.713,Z 341.972,A -85,B 0,C 180,E1 -7172.681,E2 -7172.681} C_VEL
LIN {X 0,Y 474.658,Z 341.984,A -85,B 0,C 180,E1 -7175.507,E2 -7175.507} C_VEL
LIN {X 0,Y 474.669,Z 341.973,A -85,B 0,C 180,E1 -7179.185,E2 -7179.185} C_VEL
LIN {X 0,Y 474.656,Z 341.984,A -85,B 0,C 180,E1 -7181.884,E2 -7181.884} C_VEL
LIN {X 0,Y 474.698,Z 341.978,A -85,B 0,C 180,E1 -7184.544,E2 -7184.544} C_VEL
LIN {X 0,Y 474.737,Z 341.968,A -85,B 0,C 180,E1 -7188.038,E2 -7188.038} C_VEL
LIN {X 0,Y 474.727,Z 341.975,A -85,B 0,C 180,E1 -7191.486,E2 -7191.486} C_VEL
LIN {X 0,Y 474.778,Z 341.972,A -85,B 0,C 180,E1 -7194.052,E2 -7194.052} C_VEL
LIN {X 0,Y 474.893,Z 341.957,A -85,B 0,C 180,E1 -7197.455,E2 -7197.455} C_VEL
LIN {X 0,Y 474.91,Z 341.955,A -85,B 0,C 180,E1 -7200,E2 -7200} C_VEL
LIN {X 0,Y 474.893,Z 341.954,A -85,B 0,C 180,E1 -7202.545,E2 -7202.545} C_VEL
LIN {X 0,Y 474.778,Z 341.971,A -85,B 0,C 180,E1 -7205.948,E2 -7205.948} C_VEL
LIN {X 0,Y 474.726,Z 341.975,A -85,B 0,C 180,E1 -7208.513,E2 -7208.513} C_VEL
LIN {X 0,Y 474.704,Z 341.978,A -85,B 0,C 180,E1 -7211.962,E2 -7211.962} C_VEL
LIN {X 0,Y 474.698,Z 341.98,A -85,B 0,C 180,E1 -7215.456,E2 -7215.456} C_VEL
LIN {X 0,Y 474.663,Z 341.984,A -85,B 0,C 180,E1 -7219.01,E2 -7219.01} C_VEL
LIN {X 0,Y 474.588,Z 341.996,A -85,B 0,C 180,E1 -7221.729,E2 -7221.729} C_VEL
LIN {X 0,Y 474.657,Z 341.989,A -85,B 0,C 180,E1 -7224.493,E2 -7224.493} C_VEL
LIN {X 0,Y 474.697,Z 341.983,A -85,B 0,C 180,E1 -7227.339,E2 -7227.339} C_VEL
LIN {X 0,Y 474.608,Z 341.994,A -85,B 0,C 180,E1 -7230.812,E2 -7230.812} C_VEL
LIN {X 0,Y 474.636,Z 341.99,A -85,B 0,C 180,E1 -7233.984,E2 -7233.984} C_VEL
LIN {X 0,Y 474.573,Z 341.998,A -85,B 0,C 180,E1 -7236.9,E2 -7236.9} C_VEL
LIN {X 0,Y 474.626,Z 341.992,A -85,B 0,C 180,E1 -7239.648,E2 -7239.648} C_VEL
LIN {X 0,Y 474.613,Z 341.987,A -85,B 0,C 180,E1 -7242.934,E2 -7242.934} C_VEL
LIN {X 0,Y 475.312,Z 345.803,A -85,B 0,C 180,E1 -7245.213,E2 -7245.213} C_VEL
LIN {X 0,Y 475.954,Z 350.236,A -85,B 0,C 180,E1 -7247.587,E2 -7247.587} C_VEL
LIN {X 0,Y 476.136,Z 354.031,A -85,B 0,C 180,E1 -7249.5,E2 -7249.5} C_VEL
LIN {X 0,Y 475.745,Z 361.308,A -85,B 0,C 180,E1 -7252.913,E2 -7252.913} C_VEL
LIN {X 0,Y 475.422,Z 368.023,A -85,B 0,C 180,E1 -7255.876,E2 -7255.876} C_VEL
LIN {X 0,Y 475.149,Z 375.549,A -85,B 0,C 180,E1 -7259.08,E2 -7259.08} C_VEL
LIN {X 0,Y 474.877,Z 381.996,A -85,B 0,C 180,E1 -7261.733,E2 -7261.733} C_VEL
LIN {X 0,Y 474.654,Z 389.016,A -85,B 0,C 180,E1 -7264.582,E2 -7264.582} C_VEL
LIN {X 0,Y 474.401,Z 397.029,A -85,B 0,C 180,E1 -7267.805,E2 -7267.805} C_VEL
LIN {X 0,Y 474.349,Z 398.887,A -85,B 0,C 180,E1 -7268.549,E2 -7268.549} C_VEL
LIN {X 0,Y 478.213,Z 415.713,A -85,B 0,C 180,E1 -7269.076,E2 -7269.076} C_VEL
LIN {X 0,Y 480.251,Z 425.677,A -85,B 0,C 180,E1 -7269.468,E2 -7269.468} C_VEL
LIN {X 0,Y 479.714,Z 439.358,A -85,B 0,C 180,E1 -7269.989,E2 -7269.989} C_VEL
LIN {X 0,Y 478.951,Z 454.053,A -85,B 0,C 180,E1 -7270.722,E2 -7270.722} C_VEL
LIN {X 0,Y 478.157,Z 467.599,A -85,B 0,C 180,E1 -7271.579,E2 -7271.579} C_VEL
LIN {X 0,Y 477.296,Z 481.399,A -85,B 0,C 180,E1 -7272.652,E2 -7272.652} C_VEL
LIN {X 0,Y 476.567,Z 493.905,A -85,B 0,C 180,E1 -7273.839,E2 -7273.839} C_VEL
LIN {X 0,Y 475.721,Z 506.171,A -85,B 0,C 180,E1 -7275.236,E2 -7275.236} C_VEL
LIN {X 0,Y 475.061,Z 517.088,A -85,B 0,C 180,E1 -7276.744,E2 -7276.744} C_VEL
LIN {X 0,Y 474.627,Z 526.191,A -85,B 0,C 180,E1 -7278.253,E2 -7278.253} C_VEL
LIN {X 0,Y 474.263,Z 533.743,A -85,B 0,C 180,E1 -7279.757,E2 -7279.757} C_VEL
LIN {X 0,Y 474.002,Z 540.795,A -85,B 0,C 180,E1 -7281.474,E2 -7281.474} C_VEL
LIN {X 0,Y 473.887,Z 546.345,A -85,B 0,C 180,E1 -7283.187,E2 -7283.187} C_VEL
LIN {X 0,Y 473.787,Z 550.541,A -85,B 0,C 180,E1 -7284.894,E2 -7284.894} C_VEL
LIN {X 0,Y 473.797,Z 553.486,A -85,B 0,C 180,E1 -7286.599,E2 -7286.599} C_VEL
LIN {X 0,Y 473.748,Z 555.24,A -85,B 0,C 180,E1 -7288.3,E2 -7288.3} C_VEL
LIN {X 0,Y 473.666,Z 555.837,A -85,B 0,C 180,E1 -7290,E2 -7290} C_VEL
LIN {X 0,Y 473.748,Z 555.237,A -85,B 0,C 180,E1 -7291.701,E2 -7291.701} C_VEL
LIN {X 0,Y 473.797,Z 553.48,A -85,B 0,C 180,E1 -7293.402,E2 -7293.402} C_VEL
LIN {X 0,Y 473.79,Z 550.537,A -85,B 0,C 180,E1 -7295.107,E2 -7295.107} C_VEL
LIN {X 0,Y 473.895,Z 546.347,A -85,B 0,C 180,E1 -7296.814,E2 -7296.814} C_VEL
LIN {X 0,Y 474.002,Z 540.793,A -85,B 0,C 180,E1 -7298.527,E2 -7298.527} C_VEL
LIN {X 0,Y 474.263,Z 533.733,A -85,B 0,C 180,E1 -7300.243,E2 -7300.243} C_VEL
LIN {X 0,Y 474.643,Z 526.184,A -85,B 0,C 180,E1 -7301.748,E2 -7301.748} C_VEL
LIN {X 0,Y 475.062,Z 517.085,A -85,B 0,C 180,E1 -7303.256,E2 -7303.256} C_VEL
LIN {X 0,Y 475.714,Z 506.165,A -85,B 0,C 180,E1 -7304.765,E2 -7304.765} C_VEL
LIN {X 0,Y 476.514,Z 493.901,A -85,B 0,C 180,E1 -7306.164,E2 -7306.164} C_VEL
LIN {X 0,Y 477.308,Z 481.402,A -85,B 0,C 180,E1 -7307.348,E2 -7307.348} C_VEL
LIN {X 0,Y 478.15,Z 467.585,A -85,B 0,C 180,E1 -7308.422,E2 -7308.422} C_VEL
LIN {X 0,Y 478.955,Z 454.03,A -85,B 0,C 180,E1 -7309.279,E2 -7309.279} C_VEL
LIN {X 0,Y 479.682,Z 439.374,A -85,B 0,C 180,E1 -7310.012,E2 -7310.012} C_VEL
LIN {X 0,Y 480.177,Z 424.839,A -85,B 0,C 180,E1 -7310.565,E2 -7310.565} C_VEL
LIN {X 0,Y 476.717,Z 408.77,A -85,B 0,C 180,E1 -7311.161,E2 -7311.161} C_VEL
LIN {X 0,Y 474.364,Z 398.833,A -85,B 0,C 180,E1 -7311.471,E2 -7311.471} C_VEL
LIN {X 0,Y 474.597,Z 390.136,A -85,B 0,C 180,E1 -7314.958,E2 -7314.958} C_VEL
LIN {X 0,Y 474.821,Z 383.142,A -85,B 0,C 180,E1 -7317.791,E2 -7317.791} C_VEL
LIN {X 0,Y 475.067,Z 377.244,A -85,B 0,C 180,E1 -7320.198,E2 -7320.198} C_VEL
LIN {X 0,Y 475.336,Z 370.167,A -85,B 0,C 180,E1 -7323.166,E2 -7323.166} C_VEL
LIN {X 0,Y 475.671,Z 363.173,A -85,B 0,C 180,E1 -7326.228,E2 -7326.228} C_VEL
LIN {X 0,Y 475.962,Z 356.25,A -85,B 0,C 180,E1 -7329.415,E2 -7329.415} C_VEL
LIN {X 0,Y 476.091,Z 351.689,A -85,B 0,C 180,E1 -7331.628,E2 -7331.628} C_VEL
LIN {X 0,Y 475.515,Z 347.181,A -85,B 0,C 180,E1 -7334,E2 -7334} C_VEL
LIN {X 0,Y 474.613,Z 341.992,A -85,B 0,C 180,E1 -7336.994,E2 -7336.994} C_VEL
LIN {X 0,Y 474.619,Z 341.99,A -85,B 0,C 180,E1 -7339.342,E2 -7339.342} C_VEL
LIN {X 0,Y 474.613,Z 341.994,A -85,B 0,C 180,E1 -7341.704,E2 -7341.704} C_VEL
LIN {X 0,Y 474.633,Z 341.993,A -85,B 0,C 180,E1 -7344.726,E2 -7344.726} C_VEL
LIN {X 0,Y 474.638,Z 341.99,A -85,B 0,C 180,E1 -7347.788,E2 -7347.788} C_VEL
LIN {X 0,Y 474.627,Z 341.992,A -85,B 0,C 180,E1 -7350.885,E2 -7350.885} C_VEL
LIN {X 0,Y 474.661,Z 341.986,A -85,B 0,C 180,E1 -7353.629,E2 -7353.629} C_VEL
LIN {X 0,Y 474.638,Z 341.988,A -85,B 0,C 180,E1 -7356.642,E2 -7356.642} C_VEL
LIN {X 0,Y 474.658,Z 341.988,A -85,B 0,C 180,E1 -7360.09,E2 -7360.09} C_VEL
LIN {X 0,Y 474.654,Z 341.987,A -85,B 0,C 180,E1 -7362.775,E2 -7362.775} C_VEL
LIN {X 0,Y 474.652,Z 341.986,A -85,B 0,C 180,E1 -7365.421,E2 -7365.421} C_VEL
LIN {X 0,Y 474.708,Z 341.98,A -85,B 0,C 180,E1 -7368.038,E2 -7368.038} C_VEL
LIN {X 0,Y 474.731,Z 341.976,A -85,B 0,C 180,E1 -7371.487,E2 -7371.487} C_VEL
LIN {X 0,Y 474.782,Z 341.97,A -85,B 0,C 180,E1 -7374.053,E2 -7374.053} C_VEL
LIN {X 0,Y 474.898,Z 341.954,A -85,B 0,C 180,E1 -7377.456,E2 -7377.456} C_VEL
LIN {X 0,Y 474.915,Z 341.954,A -85,B 0,C 180,E1 -7380,E2 -7380} C_VEL
LIN {X 0,Y 474.897,Z 341.955,A -85,B 0,C 180,E1 -7382.545,E2 -7382.545} C_VEL
LIN {X 0,Y 474.783,Z 341.97,A -85,B 0,C 180,E1 -7385.948,E2 -7385.948} C_VEL
LIN {X 0,Y 474.732,Z 341.975,A -85,B 0,C 180,E1 -7388.514,E2 -7388.514} C_VEL
LIN {X 0,Y 474.708,Z 341.969,A -85,B 0,C 180,E1 -7391.962,E2 -7391.962} C_VEL
LIN {X 0,Y 474.704,Z 341.978,A -85,B 0,C 180,E1 -7395.456,E2 -7395.456} C_VEL
LIN {X 0,Y 474.668,Z 341.978,A -85,B 0,C 180,E1 -7399.01,E2 -7399.01} C_VEL
LIN {X 0,Y 474.592,Z 341.988,A -85,B 0,C 180,E1 -7401.729,E2 -7401.729} C_VEL
LIN {X 0,Y 474.644,Z 341.986,A -85,B 0,C 180,E1 -7404.494,E2 -7404.494} C_VEL
LIN {X 0,Y 474.684,Z 341.974,A -85,B 0,C 180,E1 -7407.334,E2 -7407.334} C_VEL
LIN {X 0,Y 474.609,Z 341.993,A -85,B 0,C 180,E1 -7410.23,E2 -7410.23} C_VEL
LIN {X 0,Y 474.646,Z 341.981,A -85,B 0,C 180,E1 -7413.22,E2 -7413.22} C_VEL
LIN {X 0,Y 474.596,Z 341.996,A -85,B 0,C 180,E1 -7416.323,E2 -7416.323} C_VEL
LIN {X 0,Y 474.631,Z 341.99,A -85,B 0,C 180,E1 -7419.648,E2 -7419.648} C_VEL
LIN {X 0,Y 474.618,Z 341.991,A -85,B 0,C 180,E1 -7422.934,E2 -7422.934} C_VEL
LIN {X 0,Y 474.612,Z 341.993,A -85,B 0,C 180,E1 -7425.895,E2 -7425.895} C_VEL
LIN {X 0,Y 474.572,Z 341.999,A -85,B 0,C 180,E1 -7428.209,E2 -7428.209} C_VEL
LIN {X 0,Y 474.36,Z 342.025,A -85,B 0,C 180,E1 -7430.425,E2 -7430.425} C_VEL
LIN {X 0,Y 474.276,Z 342.546,A -85,B 0,C 180,E1 -7431.755,E2 -7431.755} C_VEL
LIN {X 0,Y 474.271,Z 345.099,A -85,B 0,C 180,E1 -7434.695,E2 -7434.695} C_VEL
LIN {X 0,Y 474.209,Z 347.787,A -85,B 0,C 180,E1 -7437.755,E2 -7437.755} C_VEL
LIN {X 0,Y 474.104,Z 350.726,A -85,B 0,C 180,E1 -7440.998,E2 -7440.998} C_VEL
LIN {X 0,Y 474.023,Z 353.196,A -85,B 0,C 180,E1 -7443.59,E2 -7443.59} C_VEL
LIN {X 0,Y 473.95,Z 356.42,A -85,B 0,C 180,E1 -7446.835,E2 -7446.835} C_VEL
LIN {X 0,Y 473.905,Z 358.33,A -85,B 0,C 180,E1 -7448.619,E2 -7448.619} C_VEL
LIN {X 0,Y 478.796,Z 373.826,A -85,B 0,C 180,E1 -7449.2,E2 -7449.2} C_VEL
LIN {X 0,Y 480.548,Z 380.295,A -85,B 0,C 180,E1 -7449.481,E2 -7449.481} C_VEL
LIN {X 0,Y 480.49,Z 384.336,A -85,B 0,C 180,E1 -7449.626,E2 -7449.626} C_VEL
LIN {X 0,Y 479.871,Z 390.038,A -85,B 0,C 180,E1 -7449.818,E2 -7449.818} C_VEL
LIN {X 0,Y 476.785,Z 399.13,A -85,B 0,C 180,E1 -7450.091,E2 -7450.091} C_VEL
LIN {X 0,Y 473.49,Z 408.11,A -85,B 0,C 180,E1 -7450.424,E2 -7450.424} C_VEL
LIN {X 0,Y 472.562,Z 413.419,A -85,B 0,C 180,E1 -7450.71,E2 -7450.71} C_VEL
LIN {X 0,Y 471.74,Z 427.204,A -85,B 0,C 180,E1 -7451.656,E2 -7451.656} C_VEL
LIN {X 0,Y 470.839,Z 440.07,A -85,B 0,C 180,E1 -7452.737,E2 -7452.737} C_VEL
LIN {X 0,Y 469.997,Z 451.908,A -85,B 0,C 180,E1 -7453.94,E2 -7453.94} C_VEL
LIN {X 0,Y 469.25,Z 462.679,A -85,B 0,C 180,E1 -7455.249,E2 -7455.249} C_VEL
LIN {X 0,Y 468.513,Z 473.147,A -85,B 0,C 180,E1 -7456.776,E2 -7456.776} C_VEL
LIN {X 0,Y 468.005,Z 481.837,A -85,B 0,C 180,E1 -7458.303,E2 -7458.303} C_VEL
LIN {X 0,Y 467.532,Z 488.114,A -85,B 0,C 180,E1 -7459.607,E2 -7459.607} C_VEL
LIN {X 0,Y 467.201,Z 495.015,A -85,B 0,C 180,E1 -7461.348,E2 -7461.348} C_VEL
LIN {X 0,Y 466.967,Z 500.436,A -85,B 0,C 180,E1 -7463.084,E2 -7463.084} C_VEL
LIN {X 0,Y 466.756,Z 504.532,A -85,B 0,C 180,E1 -7464.816,E2 -7464.816} C_VEL
LIN {X 0,Y 466.755,Z 507.405,A -85,B 0,C 180,E1 -7466.547,E2 -7466.547} C_VEL
LIN {X 0,Y 466.694,Z 509.139,A -85,B 0,C 180,E1 -7468.274,E2 -7468.274} C_VEL
LIN {X 0,Y 466.597,Z 509.749,A -85,B 0,C 180,E1 -7470,E2 -7470} C_VEL
LIN {X 0,Y 466.694,Z 509.19,A -85,B 0,C 180,E1 -7471.726,E2 -7471.726} C_VEL
LIN {X 0,Y 466.755,Z 507.526,A -85,B 0,C 180,E1 -7473.453,E2 -7473.453} C_VEL
LIN {X 0,Y 466.751,Z 504.719,A -85,B 0,C 180,E1 -7475.183,E2 -7475.183} C_VEL
LIN {X 0,Y 466.95,Z 500.689,A -85,B 0,C 180,E1 -7476.915,E2 -7476.915} C_VEL
LIN {X 0,Y 467.197,Z 495.345,A -85,B 0,C 180,E1 -7478.651,E2 -7478.651} C_VEL
LIN {X 0,Y 467.502,Z 488.534,A -85,B 0,C 180,E1 -7480.392,E2 -7480.392} C_VEL
LIN {X 0,Y 467.983,Z 481.2,A -85,B 0,C 180,E1 -7481.916,E2 -7481.916} C_VEL
LIN {X 0,Y 468.543,Z 472.362,A -85,B 0,C 180,E1 -7483.444,E2 -7483.444} C_VEL
LIN {X 0,Y 469.189,Z 463.342,A -85,B 0,C 180,E1 -7484.752,E2 -7484.752} C_VEL
LIN {X 0,Y 469.926,Z 452.697,A -85,B 0,C 180,E1 -7486.062,E2 -7486.062} C_VEL
LIN {X 0,Y 470.797,Z 441.141,A -85,B 0,C 180,E1 -7487.251,E2 -7487.251} C_VEL
LIN {X 0,Y 471.628,Z 428.356,A -85,B 0,C 180,E1 -7488.348,E2 -7488.348} C_VEL
LIN {X 0,Y 472.443,Z 414.323,A -85,B 0,C 180,E1 -7489.328,E2 -7489.328} C_VEL
LIN {X 0,Y 473.248,Z 399.611,A -85,B 0,C 180,E1 -7490.137,E2 -7490.137} C_VEL
LIN {X 0,Y 473.804,Z 384.806,A -85,B 0,C 180,E1 -7490.761,E2 -7490.761} C_VEL
LIN {X 0,Y 473.76,Z 381.256,A -85,B 0,C 180,E1 -7490.896,E2 -7490.896} C_VEL
LIN {X 0,Y 469.749,Z 367.642,A -85,B 0,C 180,E1 -7491.485,E2 -7491.485} C_VEL
LIN {X 0,Y 466.84,Z 358.584,A -85,B 0,C 180,E1 -7491.835,E2 -7491.835} C_VEL
LIN {X 0,Y 466.936,Z 355.455,A -85,B 0,C 180,E1 -7494.925,E2 -7494.925} C_VEL
LIN {X 0,Y 466.984,Z 352.663,A -85,B 0,C 180,E1 -7497.81,E2 -7497.81} C_VEL
LIN {X 0,Y 467.064,Z 349.811,A -85,B 0,C 180,E1 -7500.942,E2 -7500.942} C_VEL
LIN {X 0,Y 467.18,Z 346.955,A -85,B 0,C 180,E1 -7504.168,E2 -7504.168} C_VEL
LIN {X 0,Y 467.219,Z 344.395,A -85,B 0,C 180,E1 -7507.133,E2 -7507.133} C_VEL
LIN {X 0,Y 467.225,Z 343.169,A -85,B 0,C 180,E1 -7508.539,E2 -7508.539} C_VEL
LIN {X 0,Y 467.482,Z 342.879,A -85,B 0,C 180,E1 -7511.263,E2 -7511.263} C_VEL
LIN {X 0,Y 467.552,Z 342.867,A -85,B 0,C 180,E1 -7513.82,E2 -7513.82} C_VEL
LIN {X 0,Y 467.555,Z 342.872,A -85,B 0,C 180,E1 -7516.255,E2 -7516.255} C_VEL
LIN {X 0,Y 467.577,Z 342.867,A -85,B 0,C 180,E1 -7518.723,E2 -7518.723} C_VEL
LIN {X 0,Y 467.565,Z 342.869,A -85,B 0,C 180,E1 -7521.955,E2 -7521.955} C_VEL
LIN {X 0,Y 467.568,Z 342.869,A -85,B 0,C 180,E1 -7525.168,E2 -7525.168} C_VEL
LIN {X 0,Y 467.583,Z 342.864,A -85,B 0,C 180,E1 -7528.26,E2 -7528.26} C_VEL
LIN {X 0,Y 467.582,Z 342.865,A -85,B 0,C 180,E1 -7531.251,E2 -7531.251} C_VEL
LIN {X 0,Y 467.61,Z 342.858,A -85,B 0,C 180,E1 -7534.16,E2 -7534.16} C_VEL
LIN {X 0,Y 467.575,Z 342.866,A -85,B 0,C 180,E1 -7536.996,E2 -7536.996} C_VEL
LIN {X 0,Y 467.622,Z 342.848,A -85,B 0,C 180,E1 -7539.777,E2 -7539.777} C_VEL
LIN {X 0,Y 467.608,Z 342.862,A -85,B 0,C 180,E1 -7542.507,E2 -7542.507} C_VEL
LIN {X 0,Y 467.605,Z 342.858,A -85,B 0,C 180,E1 -7545.196,E2 -7545.196} C_VEL
LIN {X 0,Y 467.681,Z 342.844,A -85,B 0,C 180,E1 -7547.855,E2 -7547.855} C_VEL
LIN {X 0,Y 467.68,Z 342.854,A -85,B 0,C 180,E1 -7551.357,E2 -7551.357} C_VEL
LIN {X 0,Y 467.743,Z 342.848,A -85,B 0,C 180,E1 -7553.963,E2 -7553.963} C_VEL
LIN {X 0,Y 467.858,Z 342.833,A -85,B 0,C 180,E1 -7557.417,E2 -7557.417} C_VEL
LIN {X 0,Y 467.881,Z 342.831,A -85,B 0,C 180,E1 -7560,E2 -7560} C_VEL
LIN {X 0,Y 467.859,Z 342.831,A -85,B 0,C 180,E1 -7562.583,E2 -7562.583} C_VEL
LIN {X 0,Y 467.742,Z 342.848,A -85,B 0,C 180,E1 -7566.037,E2 -7566.037} C_VEL
LIN {X 0,Y 467.68,Z 342.853,A -85,B 0,C 180,E1 -7568.643,E2 -7568.643} C_VEL
LIN {X 0,Y 467.655,Z 342.858,A -85,B 0,C 180,E1 -7572.145,E2 -7572.145} C_VEL
LIN {X 0,Y 467.637,Z 342.859,A -85,B 0,C 180,E1 -7575.695,E2 -7575.695} C_VEL
LIN {X 0,Y 467.615,Z 342.863,A -85,B 0,C 180,E1 -7578.765,E2 -7578.765} C_VEL
LIN {X 0,Y 467.579,Z 342.867,A -85,B 0,C 180,E1 -7581.269,E2 -7581.269} C_VEL
LIN {X 0,Y 467.571,Z 342.868,A -85,B 0,C 180,E1 -7583.943,E2 -7583.943} C_VEL
LIN {X 0,Y 467.614,Z 342.863,A -85,B 0,C 180,E1 -7586.8,E2 -7586.8} C_VEL
LIN {X 0,Y 467.585,Z 342.866,A -85,B 0,C 180,E1 -7589.736,E2 -7589.736} C_VEL
LIN {X 0,Y 467.581,Z 342.867,A -85,B 0,C 180,E1 -7592.758,E2 -7592.758} C_VEL
LIN {X 0,Y 467.555,Z 342.871,A -85,B 0,C 180,E1 -7595.889,E2 -7595.889} C_VEL
LIN {X 0,Y 467.58,Z 342.866,A -85,B 0,C 180,E1 -7599.145,E2 -7599.145} C_VEL
LIN {X 0,Y 467.587,Z 342.862,A -85,B 0,C 180,E1 -7602.626,E2 -7602.626} C_VEL
LIN {X 0,Y 468.343,Z 347.132,A -85,B 0,C 180,E1 -7605.148,E2 -7605.148} C_VEL
LIN {X 0,Y 468.989,Z 351.59,A -85,B 0,C 180,E1 -7607.597,E2 -7607.597} C_VEL
LIN {X 0,Y 469.125,Z 356.132,A -85,B 0,C 180,E1 -7609.896,E2 -7609.896} C_VEL
LIN {X 0,Y 468.709,Z 363.026,A -85,B 0,C 180,E1 -7613.147,E2 -7613.147} C_VEL
LIN {X 0,Y 468.437,Z 368.498,A -85,B 0,C 180,E1 -7615.606,E2 -7615.606} C_VEL
